C01810=1025.113,288.179,370.569,170.460,47.776,159.220
C01811=1025.106,287.931,370.600,170.455,47.778,159.220
C01812=1025.099,287.683,370.631,170.450,47.780,159.220
C01813=1025.092,287.435,370.663,170.446,47.782,159.220
C01814=1025.086,287.188,370.694,170.441,47.784,159.219
C01815=1025.080,286.940,370.725,170.437,47.786,159.219
C01816=1025.073,286.692,370.757,170.432,47.788,159.219
C01817=1025.066,286.444,370.788,170.428,47.790,159.219
C01818=1025.059,286.196,370.820,170.423,47.792,159.219
C01819=1025.053,285.948,370.851,170.419,47.794,159.219
C01820=1025.046,285.700,370.883,170.414,47.796,159.219
C01821=1025.039,285.452,370.914,170.410,47.798,159.218
C01822=1025.033,285.204,370.945,170.405,47.800,159.218
C01823=1025.026,284.956,370.976,170.400,47.802,159.218
C01824=1025.019,284.708,371.008,170.397,47.804,159.218
C01825=1025.013,284.461,371.039,170.392,47.806,159.218
C01826=1025.006,284.213,371.069,170.387,47.808,159.218
C01827=1024.999,283.965,371.100,170.382,47.810,159.217
C01828=1024.993,283.717,371.132,170.378,47.812,159.217
C01829=1024.986,283.468,371.162,170.374,47.814,159.217
C01830=1024.979,283.220,371.194,170.369,47.816,159.217
C01831=1024.973,282.973,371.225,170.365,47.818,159.217
C01832=1024.966,282.724,371.256,170.360,47.821,159.217
C01833=1024.959,282.477,371.286,170.356,47.823,159.217
C01834=1024.953,282.229,371.318,170.352,47.825,159.217
C01835=1024.946,281.981,371.349,170.347,47.827,159.216
C01836=1024.940,281.733,371.380,170.342,47.829,159.216
C01837=1024.933,281.484,371.411,170.339,47.831,159.216
C01838=1024.927,281.237,371.442,170.334,47.833,159.216
C01839=1024.920,280.989,371.473,170.329,47.835,159.216
C01840=1024.913,280.741,371.503,170.325,47.838,159.216
C01841=1024.906,280.493,371.535,170.321,47.839,159.216
C01842=1024.901,280.245,371.565,170.316,47.841,159.215
C01843=1024.894,279.997,371.597,170.312,47.844,159.216
C01844=1024.887,279.749,371.627,170.307,47.846,159.215
C01845=1024.880,279.501,371.658,170.303,47.848,159.215
C01846=1024.874,279.253,371.688,170.299,47.850,159.215
C01847=1024.867,279.005,371.720,170.294,47.853,159.215
C01848=1024.861,278.757,371.751,170.290,47.855,159.215
C01849=1024.851,278.345,371.802,170.283,47.858,159.215
C01850=1024.839,277.933,371.853,170.276,47.862,159.215
C01851=1024.829,277.521,371.904,170.269,47.866,159.215
C01852=1024.818,277.109,371.955,170.261,47.870,159.214
C01853=1024.811,276.860,371.985,170.256,47.872,159.214
C01854=1024.805,276.613,372.016,170.253,47.874,159.214
C01855=1024.798,276.365,372.047,170.248,47.876,159.214
C01856=1024.791,276.116,372.077,170.244,47.879,159.214
C01857=1024.785,275.869,372.107,170.239,47.881,159.214
C01858=1024.779,275.620,372.138,170.236,47.884,159.214
C01859=1024.771,275.372,372.169,170.231,47.886,159.214
C01860=1024.765,275.125,372.199,170.227,47.888,159.214
C01861=1024.758,274.876,372.229,170.222,47.891,159.214
C01862=1024.753,274.629,372.260,170.219,47.893,159.214
C01863=1024.746,274.380,372.290,170.214,47.895,159.214
C01864=1024.739,274.132,372.320,170.209,47.898,159.214
C01865=1024.733,273.884,372.351,170.206,47.900,159.213
C01866=1024.726,273.636,372.381,170.201,47.902,159.213
C01867=1024.720,273.388,372.411,170.197,47.905,159.213
C01868=1024.713,273.140,372.442,170.192,47.907,159.213
C01869=1024.706,272.892,372.473,170.189,47.910,159.213
C01870=1024.700,272.644,372.502,170.184,47.912,159.213
C01871=1024.693,272.396,372.533,170.180,47.914,159.213
C01872=1024.687,272.148,372.563,170.176,47.917,159.213
C01873=1024.681,271.899,372.593,170.172,47.919,159.213
C01874=1024.674,271.652,372.623,170.167,47.922,159.213
C01875=1024.668,271.403,372.653,170.163,47.924,159.213
C01876=1024.661,271.156,372.683,170.159,47.926,159.213
C01877=1024.655,270.907,372.714,170.155,47.929,159.213
C01878=1024.648,270.659,372.744,170.150,47.932,159.213
C01879=1024.642,270.411,372.774,170.147,47.934,159.213
C01880=1024.635,270.163,372.805,170.142,47.936,159.213
C01881=1024.629,269.915,372.835,170.138,47.939,159.213
C01882=1024.622,269.667,372.864,170.134,47.941,159.213
C01883=1024.615,269.419,372.894,170.130,47.944,159.213
C01884=1024.610,269.171,372.924,170.125,47.946,159.213
C01885=1024.602,268.923,372.954,170.121,47.949,159.213
C01886=1024.596,268.675,372.984,170.118,47.952,159.213
C01887=1024.590,268.426,373.014,170.113,47.954,159.213
C01888=1024.583,268.179,373.044,170.109,47.957,159.213
C01889=1024.576,267.930,373.074,170.105,47.959,159.213
C01890=1024.570,267.682,373.104,170.101,47.962,159.213
C01891=1024.563,267.434,373.134,170.096,47.964,159.213
C01892=1024.557,267.186,373.164,170.093,47.967,159.213
C01893=1024.550,266.937,373.193,170.088,47.969,159.213
C01894=1024.544,266.689,373.223,170.084,47.972,159.213
C01895=1024.538,266.442,373.253,170.080,47.975,159.213
C01896=1024.531,266.193,373.283,170.076,47.977,159.213
C01897=1024.525,265.945,373.313,170.072,47.980,159.213
C01898=1024.518,265.696,373.342,170.067,47.983,159.213
C01899=1024.511,265.449,373.372,170.064,47.985,159.213
C01900=1024.505,265.201,373.401,170.060,47.988,159.213
C01901=1024.498,264.953,373.431,170.055,47.991,159.213
C01902=1024.492,264.704,373.460,170.052,47.993,159.213
C01903=1024.485,264.456,373.491,170.047,47.996,159.213
C01904=1024.479,264.208,373.520,170.043,47.999,159.213
C01905=1024.468,263.801,373.569,170.036,48.003,159.213
C01906=1024.458,263.393,373.617,170.030,48.008,159.213
C01907=1024.448,262.986,373.665,170.023,48.012,159.213
C01908=1024.436,262.578,373.714,170.016,48.016,159.213
C01909=1024.430,262.330,373.744,170.013,48.019,159.213
C01910=1024.424,262.082,373.773,170.009,48.022,159.213
C01911=1024.417,261.834,373.803,170.004,48.025,159.213
C01912=1024.411,261.586,373.832,170.001,48.027,159.214
C01913=1024.404,261.337,373.861,169.996,48.030,159.214
C01914=1024.398,261.090,373.891,169.992,48.033,159.214
C01915=1024.391,260.841,373.920,169.989,48.035,159.214
C01916=1024.385,260.593,373.950,169.984,48.038,159.214
C01917=1024.378,260.345,373.979,169.980,48.041,159.214
C01918=1024.372,260.096,374.008,169.977,48.044,159.214
C01919=1024.365,259.848,374.038,169.972,48.047,159.214
C01920=1024.358,259.601,374.066,169.968,48.050,159.214
C01921=1024.352,259.352,374.095,169.964,48.053,159.214
C01922=1024.345,259.104,374.125,169.960,48.055,159.214
C01923=1024.339,258.856,374.154,169.956,48.059,159.214
C01924=1024.332,258.608,374.182,169.952,48.061,159.214
C01925=1024.325,258.360,374.211,169.948,48.065,159.214
C01926=1024.319,258.111,374.241,169.945,48.067,159.215
C01927=1024.312,257.863,374.270,169.940,48.070,159.215
C01928=1024.305,257.615,374.298,169.936,48.073,159.215
C01929=1024.298,257.366,374.327,169.933,48.076,159.215
C01930=1024.292,257.118,374.356,169.929,48.079,159.215
C01931=1024.286,256.870,374.385,169.924,48.082,159.215
C01932=1024.279,256.622,374.414,169.920,48.085,159.215
C01933=1024.273,256.374,374.443,169.917,48.088,159.215
C01934=1024.266,256.125,374.472,169.913,48.091,159.215
C01935=1024.259,255.876,374.500,169.908,48.094,159.215
C01936=1024.253,255.628,374.529,169.905,48.097,159.215
C01937=1024.247,255.380,374.558,169.901,48.100,159.216
C01938=1024.240,255.132,374.587,169.896,48.103,159.216
C01939=1024.233,254.884,374.616,169.892,48.106,159.216
C01940=1024.227,254.635,374.645,169.889,48.109,159.216
C01941=1024.220,254.387,374.674,169.885,48.112,159.216
C01942=1024.214,254.139,374.703,169.881,48.115,159.216
C01943=1024.207,253.891,374.731,169.877,48.118,159.216
C01944=1024.201,253.643,374.760,169.873,48.121,159.217
C01945=1024.194,253.394,374.789,169.869,48.124,159.217
C01946=1024.187,253.146,374.818,169.866,48.127,159.217
C01947=1024.181,252.898,374.847,169.862,48.130,159.217
C01948=1024.175,252.649,374.875,169.857,48.133,159.217
C01949=1024.169,252.401,374.904,169.854,48.136,159.217
C01950=1024.162,252.153,374.933,169.850,48.139,159.217
C01951=1024.156,251.904,374.961,169.846,48.143,159.217
C01952=1024.150,251.656,374.990,169.842,48.145,159.217
C01953=1024.143,251.408,375.018,169.839,48.149,159.218
C01954=1024.136,251.160,375.047,169.834,48.151,159.218
C01955=1024.131,250.912,375.076,169.830,48.155,159.218
C01956=1024.124,250.663,375.105,169.827,48.158,159.218
C01957=1024.117,250.415,375.134,169.823,48.161,159.218
C01958=1024.111,250.166,375.162,169.819,48.164,159.218
C01959=1024.105,249.918,375.191,169.815,48.167,159.218
C01960=1024.098,249.670,375.219,169.811,48.170,159.218
C01961=1024.088,249.261,375.266,169.805,48.176,159.219
C01962=1024.077,248.852,375.313,169.799,48.180,159.219
C01963=1024.067,248.442,375.361,169.792,48.186,159.219
C01964=1024.057,248.034,375.407,169.786,48.191,159.219
C01965=1024.050,247.786,375.436,169.783,48.194,159.220
C01966=1024.044,247.538,375.465,169.778,48.197,159.220
C01967=1024.037,247.289,375.493,169.775,48.200,159.220
C01968=1024.031,247.041,375.522,169.771,48.203,159.220
C01969=1024.025,246.792,375.550,169.767,48.207,159.220
C01970=1024.018,246.544,375.579,169.764,48.209,159.220
C01971=1024.012,246.296,375.607,169.760,48.213,159.221
C01972=1024.006,246.047,375.636,169.756,48.216,159.221
C01973=1023.999,245.799,375.664,169.753,48.219,159.221
C01974=1023.993,245.551,375.693,169.748,48.222,159.221
C01975=1023.987,245.302,375.721,169.744,48.225,159.221
C01976=1023.981,245.053,375.749,169.741,48.228,159.221
C01977=1023.975,244.806,375.778,169.737,48.232,159.222
C01978=1023.969,244.558,375.806,169.734,48.235,159.222
C01979=1023.963,244.309,375.835,169.729,48.238,159.222
C01980=1023.956,244.061,375.863,169.725,48.241,159.222
C01981=1023.950,243.812,375.891,169.722,48.244,159.222
C01982=1023.943,243.564,375.919,169.718,48.248,159.222
C01983=1023.937,243.316,375.948,169.714,48.251,159.223
C01984=1023.930,243.067,375.975,169.711,48.254,159.223
C01985=1023.925,242.820,376.004,169.707,48.258,159.223
C01986=1023.918,242.571,376.032,169.703,48.261,159.223
C01987=1023.912,242.323,376.060,169.700,48.264,159.223
C01988=1023.905,242.074,376.088,169.696,48.268,159.224
C01989=1023.899,241.826,376.116,169.692,48.271,159.224
C01990=1023.893,241.578,376.145,169.689,48.274,159.224
C01991=1023.886,241.329,376.172,169.685,48.278,159.224
C01992=1023.880,241.080,376.201,169.681,48.281,159.224
C01993=1023.874,240.833,376.228,169.678,48.284,159.225
C01994=1023.867,240.584,376.256,169.674,48.288,159.225
C01995=1023.861,240.335,376.284,169.670,48.291,159.225
C01996=1023.855,240.087,376.312,169.667,48.294,159.225
C01997=1023.848,239.839,376.341,169.662,48.298,159.225
C01998=1023.842,239.591,376.368,169.658,48.301,159.226
C01999=1023.836,239.343,376.396,169.655,48.304,159.226
C02000=1023.829,239.094,376.424,169.652,48.309,159.226
C02001=1023.822,238.846,376.452,169.648,48.312,159.226
C02002=1023.816,238.597,376.480,169.645,48.315,159.227
C02003=1023.810,238.349,376.508,169.640,48.319,159.227
C02004=1023.804,238.100,376.534,169.637,48.323,159.227
C02005=1023.797,237.852,376.562,169.634,48.326,159.227
C02006=1023.790,237.603,376.590,169.630,48.329,159.228
C02007=1023.784,237.355,376.617,169.626,48.333,159.228
C02008=1023.778,237.107,376.645,169.623,48.336,159.228
C02009=1023.772,236.858,376.673,169.619,48.340,159.228
C02010=1023.765,236.610,376.701,169.615,48.343,159.228
C02011=1023.758,236.362,376.729,169.611,48.347,159.229
C02012=1023.752,236.113,376.756,169.608,48.351,159.229
C02013=1023.746,235.865,376.783,169.604,48.354,159.229
C02014=1023.739,235.616,376.811,169.600,48.358,159.229
C02015=1023.733,235.368,376.838,169.597,48.361,159.230
C02016=1023.726,235.119,376.866,169.593,48.365,159.230
C02017=1023.716,234.704,376.912,169.587,48.370,159.230
C02018=1023.705,234.289,376.958,169.581,48.377,159.231
C02019=1023.694,233.874,377.004,169.574,48.383,159.231
C02020=1023.684,233.458,377.050,169.569,48.388,159.232
C02021=1023.678,233.210,377.077,169.565,48.392,159.232
C02022=1023.671,232.962,377.105,169.561,48.396,159.232
C02023=1023.665,232.713,377.132,169.559,48.400,159.233
C02024=1023.658,232.464,377.160,169.555,48.403,159.233
C02025=1023.652,232.217,377.187,169.550,48.407,159.233
C02026=1023.646,231.968,377.214,169.548,48.410,159.233
C02027=1023.639,231.719,377.242,169.544,48.414,159.234
C02028=1023.633,231.471,377.269,169.540,48.418,159.234
C02029=1023.627,231.222,377.296,169.536,48.421,159.234
C02030=1023.620,230.975,377.324,169.533,48.425,159.234
C02031=1023.614,230.726,377.351,169.529,48.429,159.235
C02032=1023.607,230.477,377.378,169.525,48.432,159.235
C02033=1023.601,230.229,377.406,169.522,48.436,159.235
C02034=1023.595,229.980,377.433,169.518,48.439,159.235
C02035=1023.588,229.732,377.461,169.515,48.444,159.236
C02036=1023.582,229.484,377.487,169.512,48.447,159.236
C02037=1023.576,229.235,377.515,169.508,48.451,159.236
C02038=1023.570,228.987,377.542,169.504,48.455,159.237
C02039=1023.563,228.738,377.569,169.501,48.458,159.237
C02040=1023.557,228.489,377.596,169.497,48.462,159.237
C02041=1023.551,228.241,377.624,169.493,48.466,159.238
C02042=1023.545,227.992,377.651,169.491,48.470,159.238
C02043=1023.538,227.745,377.678,169.487,48.474,159.238
C02044=1023.531,227.496,377.705,169.483,48.477,159.239
C02045=1023.525,227.247,377.732,169.479,48.481,159.239
C02046=1023.519,226.999,377.759,169.476,48.485,159.239
C02047=1023.512,226.750,377.786,169.472,48.489,159.239
C02048=1023.506,226.502,377.812,169.469,48.493,159.240
C02049=1023.499,226.254,377.840,169.466,48.496,159.240
C02050=1023.494,226.005,377.866,169.462,48.500,159.240
C02051=1023.486,225.756,377.893,169.458,48.504,159.241
C02052=1023.480,225.508,377.921,169.455,48.508,159.241
C02053=1023.474,225.260,377.947,169.452,48.512,159.242
C02054=1023.467,225.011,377.974,169.448,48.516,159.242
C02055=1023.461,224.763,378.000,169.444,48.520,159.242
C02056=1023.454,224.514,378.028,169.440,48.524,159.242
C02057=1023.448,224.266,378.054,169.438,48.528,159.243
C02058=1023.441,224.017,378.081,169.434,48.532,159.243
C02059=1023.436,223.769,378.108,169.430,48.536,159.244
C02060=1023.429,223.520,378.134,169.426,48.539,159.244
C02061=1023.423,223.272,378.161,169.423,48.543,159.244
C02062=1023.416,223.023,378.188,169.420,48.547,159.244
C02063=1023.410,222.775,378.215,169.416,48.551,159.245
C02064=1023.403,222.526,378.242,169.413,48.555,159.245
C02065=1023.397,222.278,378.268,169.410,48.559,159.246
C02066=1023.390,222.029,378.295,169.406,48.563,159.246
C02067=1023.385,221.780,378.321,169.402,48.567,159.246
C02068=1023.378,221.532,378.349,169.399,48.571,159.247
C02069=1023.371,221.284,378.375,169.395,48.575,159.247
C02070=1023.365,221.035,378.402,169.392,48.579,159.247
C02071=1023.359,220.787,378.429,169.389,48.583,159.248
C02072=1023.352,220.538,378.455,169.385,48.587,159.248
C02073=1023.347,220.326,378.478,169.382,48.590,159.248
C02074=1023.342,220.115,378.500,169.379,48.593,159.249
C02075=1023.336,219.903,378.523,169.377,48.597,159.249
C02076=1023.332,219.691,378.546,169.374,48.600,159.249
C02077=1023.326,219.481,378.569,169.371,48.604,159.249
C02078=1023.320,219.269,378.591,169.368,48.607,159.250
C02079=1023.316,219.057,378.614,169.365,48.611,159.250
C02080=1023.310,218.846,378.636,169.362,48.614,159.250
C02081=1023.304,218.597,378.663,169.358,48.618,159.251
C02082=1023.297,218.349,378.690,169.355,48.623,159.251
C02083=1023.290,218.100,378.716,169.351,48.627,159.252
C02084=1023.284,217.852,378.743,169.348,48.631,159.252
C02085=1023.278,217.603,378.768,169.345,48.635,159.252
C02086=1023.271,217.354,378.794,169.341,48.639,159.253
C02087=1023.265,217.106,378.821,169.337,48.643,159.253
C02088=1023.258,216.857,378.847,169.335,48.647,159.253
C02089=1023.252,216.609,378.873,169.331,48.651,159.254
C02090=1023.246,216.361,378.900,169.327,48.655,159.254
C02091=1023.239,216.111,378.926,169.324,48.660,159.255
C02092=1023.232,215.863,378.952,169.321,48.664,159.255
C02093=1023.226,215.614,378.979,169.317,48.668,159.255
C02094=1023.220,215.366,379.005,169.314,48.672,159.256
C02095=1023.214,215.118,379.032,169.310,48.676,159.256
C02096=1023.207,214.868,379.057,169.307,48.680,159.257
C02097=1023.200,214.620,379.083,169.304,48.685,159.257
C02098=1023.195,214.372,379.110,169.300,48.689,159.257
C02099=1023.188,214.123,379.136,169.297,48.693,159.258
C02100=1023.181,213.875,379.162,169.293,48.697,159.258
C02101=1023.176,213.626,379.188,169.290,48.701,159.259
C02102=1023.169,213.377,379.215,169.287,48.706,159.259
C02103=1023.162,213.129,379.240,169.283,48.710,159.259
C02104=1023.157,212.880,379.267,169.279,48.714,159.260
C02105=1023.150,212.632,379.293,169.277,48.718,159.260
C02106=1023.143,212.384,379.319,169.273,48.723,159.261
C02107=1023.137,212.135,379.345,169.270,48.727,159.261
C02108=1023.131,211.887,379.371,169.266,48.731,159.261
C02109=1023.125,211.637,379.398,169.263,48.735,159.262
C02110=1023.118,211.389,379.424,169.260,48.740,159.262
C02111=1023.112,211.141,379.450,169.256,48.744,159.263
C02112=1023.106,210.892,379.476,169.252,48.748,159.263
C02113=1023.099,210.643,379.502,169.250,48.752,159.264
C02114=1023.093,210.395,379.528,169.246,48.757,159.264
C02115=1023.087,210.146,379.554,169.243,48.761,159.264
C02116=1023.081,209.898,379.580,169.239,48.765,159.265
C02117=1023.074,209.649,379.606,169.237,48.770,159.265
C02118=1023.067,209.401,379.632,169.233,48.774,159.266
C02119=1023.061,209.152,379.657,169.230,48.779,159.266
C02120=1023.055,208.904,379.683,169.226,48.783,159.267
C02121=1023.048,208.655,379.709,169.223,48.788,159.267
C02122=1023.042,208.406,379.736,169.220,48.792,159.268
C02123=1023.036,208.157,379.761,169.216,48.796,159.268
C02124=1023.029,207.909,379.787,169.213,48.801,159.268
C02125=1023.023,207.661,379.812,169.209,48.805,159.269
C02126=1023.016,207.411,379.838,169.207,48.809,159.269
C02127=1023.010,207.163,379.864,169.203,48.814,159.270
C02128=1023.004,206.915,379.889,169.200,48.818,159.270
C02129=1022.997,206.667,379.915,169.196,48.823,159.271
C02130=1022.991,206.418,379.941,169.193,48.827,159.271
C02131=1022.985,206.168,379.967,169.190,48.831,159.272
C02132=1022.978,205.920,379.993,169.187,48.836,159.272
C02133=1022.968,205.500,380.036,169.181,48.844,159.273
C02134=1022.957,205.080,380.080,169.175,48.851,159.274
C02135=1022.946,204.659,380.122,169.169,48.859,159.274
C02136=1022.935,204.239,380.166,169.164,48.867,159.275
C02137=1022.911,203.207,380.265,168.742,48.769,159.192
C02138=1022.906,202.959,380.290,168.738,48.774,159.192
C02139=1022.900,202.709,380.314,168.734,48.780,159.193
C02140=1022.895,202.460,380.338,168.730,48.785,159.193
C02141=1022.889,202.212,380.361,168.725,48.790,159.194
C02142=1022.884,201.963,380.386,168.721,48.796,159.194
C02143=1022.879,201.715,380.410,168.717,48.801,159.195
C02144=1022.873,201.465,380.434,168.713,48.807,159.196
C02145=1022.867,201.216,380.458,168.708,48.812,159.196
C02146=1022.862,200.968,380.482,168.705,48.818,159.197
C02147=1022.856,200.719,380.506,168.701,48.823,159.197
C02148=1022.851,200.470,380.530,168.696,48.828,159.197
C02149=1022.845,200.222,380.553,168.692,48.834,159.198
C02150=1022.839,199.973,380.578,168.688,48.839,159.198
C02151=1022.834,199.723,380.601,168.684,48.845,159.199
C02152=1022.828,199.475,380.625,168.680,48.850,159.199
C02153=1022.823,199.226,380.649,168.675,48.856,159.200
C02154=1022.817,198.978,380.672,168.671,48.861,159.200
C02155=1022.812,198.729,380.695,168.667,48.867,159.201
C02156=1022.806,198.479,380.720,168.663,48.873,159.202
C02157=1022.800,198.230,380.743,168.659,48.878,159.202
C02158=1022.795,197.982,380.767,168.655,48.884,159.203
C02159=1022.789,197.733,380.790,168.651,48.890,159.203
C02160=1022.783,197.485,380.814,168.646,48.895,159.204
C02161=1022.778,197.236,380.837,168.642,48.901,159.204
C02162=1022.772,196.987,380.861,168.638,48.906,159.205
C02163=1022.766,196.738,380.884,168.634,48.912,159.205
C02164=1022.761,196.489,380.907,168.630,48.917,159.206
C02165=1022.754,196.240,380.931,168.625,48.923,159.206
C02166=1022.749,195.991,380.955,168.621,48.928,159.207
C02167=1022.743,195.743,380.979,168.617,48.934,159.207
C02168=1022.738,195.494,381.002,168.613,48.939,159.208
C02169=1022.733,195.245,381.025,168.609,48.945,159.208
C02170=1022.727,194.996,381.049,168.606,48.951,159.209
C02171=1022.721,194.747,381.072,168.601,48.956,159.210
C02172=1022.716,194.498,381.095,168.597,48.962,159.210
C02173=1022.710,194.250,381.119,168.593,48.968,159.211
C02174=1022.705,194.001,381.142,168.589,48.973,159.211
C02175=1022.699,193.752,381.165,168.585,48.979,159.212
C02176=1022.693,193.504,381.189,168.581,48.985,159.212
C02177=1022.688,193.254,381.213,168.576,48.990,159.213
C02178=1022.682,193.005,381.236,168.572,48.996,159.213
C02179=1022.677,192.757,381.258,168.568,49.001,159.214
C02180=1022.671,192.508,381.283,168.565,49.006,159.214
C02181=1022.666,192.259,381.306,168.561,49.012,159.215
C02182=1022.660,192.010,381.329,168.557,49.018,159.216
C02183=1022.655,191.761,381.352,168.553,49.023,159.216
C02184=1022.649,191.512,381.375,168.548,49.029,159.217
C02185=1022.644,191.263,381.399,168.544,49.035,159.217
C02186=1022.638,191.015,381.422,168.541,49.040,159.218
C02187=1022.632,190.766,381.445,168.537,49.046,159.218
C02188=1022.627,190.516,381.469,168.533,49.052,159.219
C02189=1022.622,190.268,381.492,168.529,49.057,159.219
C02190=1022.616,190.019,381.515,168.525,49.063,159.220
C02191=1022.611,189.771,381.539,168.521,49.068,159.221
C02192=1022.606,189.522,381.562,168.517,49.073,159.221
C02193=1022.600,189.273,381.584,168.513,49.079,159.222
C02194=1022.595,189.024,381.608,168.509,49.085,159.222
C02195=1022.589,188.775,381.631,168.505,49.090,159.223
C02196=1022.583,188.526,381.654,168.501,49.096,159.223
C02197=1022.578,188.277,381.677,168.498,49.102,159.224
C02198=1022.572,187.995,381.704,168.493,49.108,159.224
C02199=1022.566,187.713,381.730,168.488,49.115,159.225
C02200=1022.560,187.431,381.756,168.484,49.121,159.226
C02201=1022.554,187.150,381.782,168.479,49.128,159.226
C02202=1022.548,186.901,381.805,168.476,49.132,159.227
C02203=1022.543,186.652,381.828,168.472,49.138,159.227
C02204=1022.538,186.403,381.851,168.468,49.144,159.228
C02205=1022.532,186.154,381.874,168.464,49.149,159.228
C02206=1022.527,185.905,381.898,168.461,49.155,159.229
C02207=1022.522,185.656,381.920,168.457,49.161,159.230
C02208=1022.516,185.408,381.943,168.453,49.167,159.230
C02209=1022.511,185.158,381.967,168.448,49.172,159.231
C02210=1022.505,184.909,381.990,168.445,49.177,159.231
C02211=1022.500,184.661,382.012,168.441,49.183,159.232
C02212=1022.495,184.412,382.036,168.437,49.189,159.232
C02213=1022.489,184.163,382.059,168.434,49.194,159.233
C02214=1022.484,183.914,382.082,168.430,49.200,159.234
C02215=1022.479,183.664,382.105,168.426,49.206,159.234
C02216=1022.474,183.416,382.127,168.421,49.211,159.235
C02217=1022.468,183.167,382.150,168.419,49.217,159.235
C02218=1022.463,182.918,382.174,168.414,49.223,159.236
C02219=1022.457,182.669,382.197,168.410,49.228,159.236
C02220=1022.452,182.421,382.219,168.407,49.233,159.237
C02221=1022.447,182.172,382.241,168.403,49.239,159.238
C02222=1022.441,181.923,382.264,168.399,49.245,159.238
C02223=1022.436,181.673,382.287,168.395,49.251,159.239
C02224=1022.430,181.424,382.310,168.391,49.257,159.239
C02225=1022.424,181.176,382.331,168.388,49.263,159.240
C02226=1022.419,180.927,382.354,168.384,49.269,159.241
C02227=1022.413,180.678,382.377,168.380,49.274,159.241
C02228=1022.407,180.429,382.398,168.376,49.280,159.242
C02229=1022.402,180.181,382.421,168.372,49.286,159.242
C02230=1022.396,179.931,382.443,168.369,49.292,159.243
C02231=1022.391,179.682,382.466,168.366,49.298,159.244
C02232=1022.384,179.433,382.488,168.362,49.304,159.244
C02233=1022.380,179.184,382.510,168.358,49.310,159.245
C02234=1022.374,178.935,382.533,168.354,49.316,159.246
C02235=1022.368,178.686,382.554,168.351,49.322,159.246
C02236=1022.362,178.437,382.577,168.347,49.328,159.247
C02237=1022.357,178.188,382.599,168.343,49.334,159.247
C02238=1022.351,177.940,382.621,168.339,49.339,159.248
C02239=1022.345,177.690,382.644,168.336,49.345,159.249
C02240=1022.340,177.442,382.666,168.332,49.351,159.249
C02241=1022.334,177.193,382.688,168.328,49.357,159.250
C02242=1022.329,176.943,382.710,168.324,49.363,159.250
C02243=1022.323,176.695,382.733,168.321,49.368,159.251
C02244=1022.318,176.446,382.755,168.317,49.374,159.252
C02245=1022.312,176.196,382.776,168.313,49.380,159.252
C02246=1022.307,175.948,382.799,168.309,49.386,159.253
C02247=1022.301,175.699,382.821,168.306,49.392,159.253
C02248=1022.295,175.449,382.843,168.302,49.398,159.254
C02249=1022.290,175.201,382.866,168.298,49.404,159.255
C02250=1022.285,174.952,382.888,168.295,49.410,159.256
C02251=1022.279,174.703,382.909,168.291,49.416,159.256
C02252=1022.273,174.454,382.932,168.287,49.422,159.257
C02253=1022.268,174.205,382.954,168.283,49.428,159.257
C02254=1022.262,173.956,382.975,168.280,49.433,159.258
C02255=1022.257,173.707,382.998,168.276,49.439,159.259
C02256=1022.252,173.459,383.020,168.272,49.445,159.259
C02257=1022.246,173.209,383.042,168.269,49.451,159.260
C02258=1022.240,172.960,383.064,168.265,49.457,159.260
C02259=1022.235,172.712,383.087,168.261,49.463,159.261
C02260=1022.229,172.462,383.108,168.258,49.468,159.262
C02261=1022.224,172.214,383.130,168.254,49.474,159.262
C02262=1022.215,171.810,383.166,168.249,49.484,159.263
C02263=1022.207,171.405,383.202,168.243,49.493,159.264
C02264=1022.199,171.076,383.231,168.238,49.501,159.265
C02265=1022.192,170.746,383.260,168.234,49.509,159.266
C02266=1022.185,170.418,383.289,168.228,49.517,159.267
C02267=1022.178,170.088,383.319,168.224,49.525,159.268
C02268=1022.172,169.839,383.340,168.220,49.530,159.268
C02269=1022.167,169.590,383.362,168.217,49.536,159.269
C02270=1022.162,169.341,383.384,168.213,49.542,159.269
C02271=1022.156,169.092,383.406,168.209,49.548,159.270
C02272=1022.151,168.843,383.428,168.206,49.554,159.271
C02273=1022.145,168.594,383.450,168.202,49.560,159.271
C02274=1022.140,168.345,383.472,168.199,49.565,159.272
C02275=1022.134,168.096,383.494,168.195,49.571,159.273
C02276=1022.129,167.847,383.515,168.191,49.577,159.273
C02277=1022.124,167.599,383.537,168.189,49.583,159.274
C02278=1022.118,167.349,383.559,168.185,49.589,159.275
C02279=1022.113,167.101,383.580,168.182,49.595,159.275
C02280=1022.107,166.851,383.603,168.178,49.601,159.276
C02281=1022.103,166.602,383.625,168.175,49.607,159.276
C02282=1022.096,166.353,383.646,168.171,49.613,159.277
C02283=1022.092,166.104,383.668,168.167,49.619,159.278
C02284=1022.087,165.855,383.690,168.164,49.624,159.278
C02285=1022.081,165.606,383.712,168.160,49.630,159.279
C02286=1022.076,165.357,383.733,168.157,49.636,159.280
C02287=1022.070,165.108,383.756,168.153,49.642,159.280
C02288=1022.065,164.859,383.777,168.150,49.647,159.281
C02289=1022.060,164.611,383.799,168.146,49.653,159.281
C02290=1022.054,164.361,383.821,168.143,49.659,159.282
C02291=1022.049,164.113,383.842,168.139,49.665,159.283
C02292=1022.044,163.864,383.864,168.136,49.671,159.283
C02293=1022.039,163.614,383.886,168.132,49.677,159.284
C02294=1022.033,163.366,383.908,168.129,49.682,159.285
C02295=1022.028,163.117,383.930,168.126,49.688,159.285
C02296=1022.022,162.868,383.951,168.123,49.695,159.286
C02297=1022.018,162.618,383.972,168.119,49.701,159.287
C02298=1022.013,162.369,383.994,168.116,49.706,159.287
C02299=1022.007,162.120,384.016,168.112,49.712,159.288
C02300=1022.002,161.871,384.038,168.109,49.718,159.288
C02301=1021.997,161.623,384.060,168.105,49.724,159.289
C02302=1021.991,161.373,384.081,168.102,49.730,159.290
C02303=1021.986,161.125,384.103,168.098,49.736,159.290
C02304=1021.981,160.875,384.124,168.095,49.741,159.291
C02305=1021.975,160.626,384.146,168.091,49.747,159.292
C02306=1021.970,160.377,384.168,168.089,49.753,159.292
C02307=1021.965,160.129,384.189,168.085,49.759,159.293
C02308=1021.960,159.880,384.211,168.082,49.764,159.293
C02309=1021.955,159.630,384.232,168.078,49.770,159.294
C02310=1021.949,159.381,384.254,168.075,49.776,159.295
C02311=1021.945,159.132,384.275,168.072,49.782,159.295
C02312=1021.939,158.884,384.297,168.068,49.788,159.296
C02313=1021.934,158.634,384.318,168.065,49.793,159.297
C02314=1021.928,158.385,384.340,168.061,49.800,159.297
C02315=1021.923,158.136,384.360,168.057,49.806,159.298
C02316=1021.917,157.887,384.382,168.055,49.812,159.299
C02317=1021.911,157.638,384.403,168.051,49.818,159.299
C02318=1021.907,157.389,384.424,168.048,49.824,159.300
C02319=1021.901,157.140,384.446,168.044,49.830,159.301
C02320=1021.895,156.891,384.466,168.041,49.836,159.301
C02321=1021.890,156.642,384.488,168.038,49.843,159.302
C02322=1021.885,156.393,384.508,168.035,49.848,159.303
C02323=1021.878,156.144,384.530,168.031,49.854,159.303
C02324=1021.873,155.861,384.553,168.027,49.861,159.304
C02325=1021.867,155.578,384.577,168.024,49.868,159.305
C02326=1021.860,155.296,384.602,168.019,49.875,159.305
C02327=1021.855,155.013,384.625,168.016,49.881,159.306
C02328=1021.849,154.765,384.646,168.013,49.888,159.307
C02329=1021.844,154.514,384.668,168.009,49.894,159.308
C02330=1021.839,154.265,384.688,168.006,49.899,159.308
C02331=1021.833,154.017,384.710,168.002,49.905,159.309
C02332=1021.828,153.768,384.730,168.000,49.912,159.310
C02333=1021.822,153.518,384.752,167.996,49.918,159.310
C02334=1021.816,153.269,384.772,167.993,49.923,159.311
C02335=1021.812,153.020,384.794,167.989,49.930,159.312
C02336=1021.806,152.771,384.815,167.986,49.936,159.312
C02337=1021.801,152.522,384.835,167.982,49.942,159.313
C02338=1021.795,152.272,384.856,167.980,49.947,159.314
C02339=1021.790,152.024,384.878,167.976,49.954,159.314
C02340=1021.784,151.775,384.898,167.973,49.960,159.315
C02341=1021.779,151.526,384.919,167.969,49.966,159.316
C02342=1021.774,151.277,384.940,167.967,49.972,159.317
C02343=1021.768,151.028,384.960,167.963,49.978,159.317
C02344=1021.762,150.778,384.981,167.960,49.984,159.318
C02345=1021.757,150.529,385.002,167.956,49.991,159.319
C02346=1021.752,150.281,385.023,167.953,49.996,159.319
C02347=1021.746,150.031,385.044,167.949,50.002,159.320
C02348=1021.741,149.782,385.064,167.947,50.009,159.321
C02349=1021.736,149.533,385.085,167.944,50.015,159.321
C02350=1021.730,149.285,385.106,167.940,50.021,159.322
C02351=1021.724,149.035,385.127,167.937,50.026,159.323
C02352=1021.719,148.786,385.148,167.934,50.033,159.323
C02353=1021.714,148.537,385.168,167.931,50.039,159.324
C02354=1021.709,148.288,385.189,167.927,50.045,159.325
C02355=1021.703,148.039,385.210,167.924,50.051,159.325
C02356=1021.698,147.790,385.231,167.920,50.057,159.326
C02357=1021.693,147.541,385.251,167.918,50.063,159.327
C02358=1021.687,147.292,385.272,167.914,50.070,159.327
C02359=1021.681,147.043,385.292,167.911,50.075,159.328
C02360=1021.676,146.794,385.312,167.908,50.081,159.329
C02361=1021.670,146.544,385.333,167.905,50.088,159.330
C02362=1021.665,146.295,385.354,167.902,50.093,159.330
C02363=1021.660,146.046,385.374,167.898,50.099,159.331
C02364=1021.654,145.797,385.395,167.895,50.106,159.332
C02365=1021.649,145.548,385.416,167.891,50.112,159.332
C02366=1021.644,145.299,385.437,167.889,50.118,159.333
C02367=1021.638,145.050,385.457,167.885,50.124,159.334
C02368=1021.633,144.800,385.476,167.882,50.130,159.334
C02369=1021.627,144.551,385.497,167.880,50.136,159.335
C02370=1021.621,144.302,385.517,167.876,50.143,159.336
C02371=1021.616,144.053,385.537,167.873,50.149,159.337
C02372=1021.611,143.804,385.558,167.869,50.155,159.337
C02373=1021.606,143.555,385.579,167.866,50.161,159.338
C02374=1021.600,143.306,385.598,167.863,50.167,159.339
C02375=1021.594,143.057,385.619,167.860,50.173,159.339
C02376=1021.589,142.808,385.640,167.857,50.180,159.340
C02377=1021.584,142.559,385.660,167.854,50.186,159.341
C02378=1021.577,142.309,385.680,167.851,50.191,159.341
C02379=1021.572,142.060,385.701,167.847,50.198,159.342
C02380=1021.567,141.811,385.722,167.844,50.204,159.343
C02381=1021.562,141.562,385.742,167.841,50.211,159.344
C02382=1021.556,141.313,385.761,167.838,50.216,159.344
C02383=1021.551,141.063,385.782,167.835,50.222,159.345
C02384=1021.545,140.814,385.802,167.832,50.229,159.346
C02385=1021.540,140.566,385.822,167.829,50.235,159.346
C02386=1021.535,140.317,385.843,167.825,50.241,159.347
C02387=1021.529,140.068,385.863,167.822,50.247,159.348
C02388=1021.523,139.784,385.886,167.819,50.254,159.348
C02389=1021.517,139.502,385.909,167.815,50.261,159.349
C02390=1021.511,139.219,385.932,167.812,50.267,159.350
C02391=1021.505,138.936,385.955,167.809,50.275,159.351
C02392=1021.500,138.687,385.976,167.805,50.281,159.352
C02393=1021.494,138.437,385.995,167.802,50.287,159.352
C02394=1021.489,138.188,386.015,167.798,50.293,159.353
C02395=1021.484,137.939,386.036,167.796,50.299,159.354
C02396=1021.478,137.690,386.055,167.793,50.305,159.354
C02397=1021.473,137.441,386.076,167.789,50.312,159.355
C02398=1021.467,137.192,386.096,167.787,50.318,159.356
C02399=1021.461,136.943,386.116,167.783,50.324,159.356
C02400=1021.456,136.693,386.136,167.780,50.330,159.357
C02401=1021.450,136.444,386.156,167.778,50.336,159.358
C02402=1021.445,136.195,386.177,167.774,50.342,159.359
C02403=1021.439,135.946,386.196,167.771,50.349,159.359
C02404=1021.434,135.696,386.216,167.767,50.355,159.360
C02405=1021.429,135.447,386.236,167.765,50.361,159.361
C02406=1021.424,135.199,386.256,167.762,50.367,159.361
C02407=1021.418,134.950,386.276,167.758,50.374,159.362
C02408=1021.412,134.700,386.295,167.756,50.380,159.363
C02409=1021.407,134.451,386.316,167.753,50.385,159.364
C02410=1021.401,134.202,386.335,167.749,50.392,159.364
C02411=1021.396,133.953,386.355,167.746,50.398,159.365
C02412=1021.390,133.703,386.375,167.743,50.405,159.366
C02413=1021.385,133.454,386.395,167.740,50.410,159.366
C02414=1021.379,133.205,386.415,167.738,50.417,159.367
C02415=1021.375,132.956,386.435,167.734,50.423,159.368
C02416=1021.369,132.707,386.455,167.731,50.429,159.369
C02417=1021.364,132.458,386.474,167.728,50.435,159.369
C02418=1021.358,132.209,386.494,167.725,50.442,159.370
C02419=1021.353,131.959,386.514,167.722,50.448,159.371
C02420=1021.347,131.710,386.534,167.719,50.453,159.371
C02421=1021.342,131.462,386.553,167.716,50.460,159.372
C02422=1021.337,131.212,386.574,167.713,50.466,159.373
C02423=1021.331,130.963,386.593,167.711,50.472,159.374
C02424=1021.326,130.714,386.613,167.707,50.479,159.374
C02425=1021.320,130.464,386.633,167.704,50.484,159.375
C02426=1021.315,130.215,386.653,167.701,50.491,159.376
C02427=1021.310,129.967,386.672,167.697,50.497,159.376
C02428=1021.304,129.717,386.691,167.695,50.503,159.377
C02429=1021.298,129.468,386.711,167.691,50.509,159.378
C02430=1021.293,129.219,386.731,167.689,50.516,159.379
C02431=1021.287,128.969,386.750,167.686,50.522,159.380
C02432=1021.282,128.720,386.770,167.682,50.528,159.380
C02433=1021.276,128.472,386.789,167.680,50.535,159.381
C02434=1021.270,128.222,386.808,167.676,50.541,159.382
C02435=1021.265,127.973,386.828,167.674,50.548,159.382
C02436=1021.259,127.723,386.847,167.671,50.554,159.383
C02437=1021.253,127.475,386.867,167.667,50.560,159.384
C02438=1021.248,127.226,386.886,167.665,50.567,159.385
C02439=1021.243,126.976,386.906,167.661,50.573,159.385
C02440=1021.237,126.727,386.925,167.659,50.579,159.386
C02441=1021.232,126.477,386.944,167.656,50.585,159.387
C02442=1021.226,126.228,386.964,167.652,50.592,159.388
C02443=1021.221,125.980,386.983,167.650,50.598,159.388
C02444=1021.215,125.730,387.002,167.647,50.604,159.389
C02445=1021.209,125.481,387.021,167.644,50.611,159.390
C02446=1021.204,125.231,387.041,167.641,50.617,159.390
C02447=1021.198,124.983,387.060,167.637,50.623,159.391
C02448=1021.193,124.734,387.080,167.635,50.629,159.392
C02449=1021.187,124.484,387.099,167.632,50.636,159.393
C02450=1021.182,124.235,387.119,167.628,50.642,159.393
C02451=1021.177,123.986,387.137,167.626,50.648,159.394
C02452=1021.170,123.702,387.160,167.622,50.655,159.395
C02453=1021.163,123.420,387.181,167.619,50.663,159.396
C02454=1021.158,123.137,387.203,167.616,50.669,159.397
C02455=1021.152,122.854,387.225,167.613,50.677,159.398
C02456=1021.146,122.604,387.244,167.609,50.683,159.398
C02457=1021.140,122.355,387.264,167.607,50.690,159.399
C02458=1021.135,122.106,387.282,167.604,50.695,159.400
C02459=1021.129,121.857,387.302,167.601,50.702,159.401
C02460=1021.123,121.608,387.322,167.597,50.708,159.401
C02461=1021.119,121.359,387.341,167.595,50.714,159.402
C02462=1021.113,121.109,387.360,167.592,50.720,159.403
C02463=1021.108,120.860,387.380,167.589,50.727,159.403
C02464=1021.103,120.611,387.399,167.586,50.733,159.404
C02465=1021.097,120.362,387.418,167.584,50.739,159.405
C02466=1021.091,120.112,387.437,167.580,50.746,159.405
C02467=1021.086,119.864,387.456,167.577,50.752,159.406
C02468=1021.080,119.614,387.475,167.574,50.758,159.407
C02469=1021.075,119.365,387.494,167.572,50.764,159.408
C02470=1021.070,119.116,387.513,167.568,50.771,159.408
C02471=1021.064,118.867,387.532,167.565,50.776,159.409
C02472=1021.059,118.617,387.552,167.563,50.783,159.410
C02473=1021.054,118.368,387.571,167.559,50.789,159.410
C02474=1021.048,118.119,387.590,167.557,50.795,159.411
C02475=1021.043,117.869,387.610,167.554,50.801,159.412
C02476=1021.038,117.621,387.629,167.552,50.808,159.413
C02477=1021.032,117.371,387.648,167.548,50.814,159.413
C02478=1021.027,117.122,387.667,167.545,50.820,159.414
C02479=1021.021,116.873,387.686,167.543,50.826,159.415
C02480=1021.015,116.624,387.705,167.540,50.833,159.416
C02481=1021.010,116.375,387.724,167.536,50.839,159.416
C02482=1021.005,116.125,387.743,167.534,50.845,159.417
C02483=1021.000,115.877,387.762,167.531,50.851,159.418
C02484=1020.994,115.627,387.781,167.528,50.857,159.419
C02485=1020.989,115.377,387.801,167.526,50.864,159.419
C02486=1020.984,115.128,387.819,167.522,50.870,159.420
C02487=1020.978,114.879,387.839,167.519,50.876,159.421
C02488=1020.973,114.630,387.858,167.517,50.882,159.421
C02489=1020.968,114.381,387.877,167.514,50.888,159.422
C02490=1020.963,114.132,387.896,167.511,50.895,159.423
C02491=1020.957,113.882,387.915,167.508,50.901,159.424
C02492=1020.952,113.634,387.934,167.505,50.906,159.424
C02493=1020.946,113.384,387.952,167.503,50.913,159.425
C02494=1020.941,113.134,387.972,167.500,50.919,159.426
C02495=1020.936,112.885,387.990,167.497,50.926,159.427
C02496=1020.930,112.636,388.010,167.494,50.931,159.427
C02497=1020.925,112.387,388.029,167.491,50.937,159.428
C02498=1020.919,112.137,388.047,167.489,50.944,159.429
C02499=1020.914,111.888,388.066,167.486,50.950,159.429
C02500=1020.909,111.639,388.085,167.482,50.957,159.430
C02501=1020.904,111.390,388.104,167.480,50.962,159.431
C02502=1020.897,111.141,388.122,167.477,50.969,159.432
C02503=1020.892,110.892,388.141,167.474,50.975,159.432
C02504=1020.887,110.642,388.160,167.471,50.982,159.433
C02505=1020.881,110.392,388.179,167.468,50.987,159.434
C02506=1020.876,110.144,388.198,167.466,50.994,159.435
C02507=1020.870,109.894,388.216,167.462,51.000,159.435
C02508=1020.865,109.645,388.234,167.460,51.007,159.436
C02509=1020.859,109.396,388.254,167.457,51.013,159.437
C02510=1020.854,109.147,388.271,167.455,51.019,159.438
C02511=1020.848,108.897,388.290,167.451,51.026,159.438
C02512=1020.843,108.648,388.309,167.448,51.032,159.439
C02513=1020.837,108.399,388.327,167.446,51.038,159.440
C02514=1020.832,108.149,388.345,167.442,51.045,159.440
C02515=1020.826,107.900,388.364,167.440,51.051,159.441
C02516=1020.820,107.617,388.385,167.437,51.058,159.442
C02517=1020.813,107.334,388.407,167.434,51.066,159.443
C02518=1020.808,107.052,388.427,167.430,51.072,159.444
C02519=1020.801,106.768,388.448,167.427,51.080,159.445
C02520=1020.796,106.519,388.467,167.424,51.086,159.445
C02521=1020.790,106.270,388.484,167.422,51.092,159.446
C02522=1020.784,106.020,388.504,167.418,51.099,159.447
C02523=1020.780,105.771,388.522,167.416,51.105,159.448
C02524=1020.773,105.522,388.540,167.414,51.112,159.448
C02525=1020.768,105.273,388.559,167.411,51.118,159.449
C02526=1020.762,105.023,388.576,167.407,51.124,159.450
C02527=1020.757,104.774,388.595,167.405,51.130,159.451
C02528=1020.752,104.525,388.614,167.402,51.137,159.451
C02529=1020.746,104.276,388.632,167.400,51.143,159.452
C02530=1020.741,104.026,388.650,167.397,51.149,159.453
C02531=1020.735,103.777,388.669,167.393,51.155,159.453
C02532=1020.730,103.528,388.687,167.391,51.162,159.454
C02533=1020.725,103.278,388.706,167.388,51.168,159.455
C02534=1020.719,103.029,388.724,167.386,51.174,159.456
C02535=1020.714,102.780,388.742,167.382,51.181,159.456
C02536=1020.708,102.531,388.761,167.380,51.187,159.457
C02537=1020.703,102.282,388.779,167.377,51.193,159.458
C02538=1020.697,102.031,388.797,167.375,51.200,159.459
C02539=1020.692,101.783,388.816,167.372,51.205,159.459
C02540=1020.687,101.534,388.834,167.369,51.212,159.460
C02541=1020.680,101.285,388.853,167.366,51.218,159.461
C02542=1020.676,101.035,388.871,167.363,51.224,159.462
C02543=1020.669,100.785,388.889,167.361,51.231,159.462
C02544=1020.664,100.537,388.908,167.358,51.237,159.463
C02545=1020.660,100.287,388.926,167.355,51.243,159.464
C02546=1020.653,100.038,388.944,167.352,51.249,159.464
C02547=1020.648,99.789,388.963,167.350,51.256,159.465
C02548=1020.643,99.540,388.980,167.347,51.262,159.466
C02549=1020.637,99.290,388.999,167.344,51.268,159.467
C02550=1020.632,99.041,389.016,167.341,51.275,159.467
C02551=1020.627,98.791,389.035,167.338,51.281,159.468
C02552=1020.621,98.542,389.053,167.336,51.287,159.469
C02553=1020.615,98.293,389.071,167.333,51.294,159.470
C02554=1020.609,98.044,389.088,167.330,51.301,159.471
C02555=1020.604,97.794,389.107,167.327,51.306,159.471
C02556=1020.599,97.545,389.124,167.325,51.313,159.472
C02557=1020.593,97.295,389.142,167.322,51.319,159.473
C02558=1020.588,97.046,389.160,167.319,51.326,159.473
C02559=1020.582,96.798,389.179,167.316,51.332,159.474
C02560=1020.576,96.548,389.197,167.314,51.338,159.475
C02561=1020.571,96.299,389.215,167.311,51.344,159.476
C02562=1020.566,96.049,389.232,167.308,51.351,159.476
C02563=1020.560,95.800,389.250,167.305,51.358,159.477
C02564=1020.554,95.551,389.268,167.303,51.364,159.478
C02565=1020.549,95.301,389.286,167.300,51.370,159.479
C02566=1020.543,95.052,389.304,167.298,51.376,159.479
C02567=1020.538,94.803,389.321,167.294,51.383,159.480
C02568=1020.533,94.553,389.340,167.291,51.389,159.481
C02569=1020.527,94.303,389.357,167.289,51.395,159.482
C02570=1020.521,94.054,389.375,167.286,51.401,159.482
C02571=1020.515,93.806,389.393,167.284,51.408,159.483
C02572=1020.511,93.557,389.412,167.280,51.414,159.484
C02573=1020.504,93.307,389.429,167.278,51.421,159.485
C02574=1020.499,93.058,389.447,167.275,51.427,159.485
C02575=1020.494,92.809,389.465,167.273,51.433,159.486
C02576=1020.489,92.560,389.483,167.270,51.439,159.487
C02577=1020.483,92.310,389.501,167.267,51.446,159.488
C02578=1020.477,92.061,389.518,167.264,51.452,159.488
C02579=1020.472,91.811,389.536,167.262,51.459,159.489
C02580=1020.465,91.528,389.556,167.259,51.466,159.490
C02581=1020.460,91.245,389.576,167.255,51.472,159.491
C02582=1020.453,90.962,389.597,167.252,51.480,159.492
C02583=1020.447,90.679,389.617,167.250,51.487,159.492
C02584=1020.442,90.430,389.635,167.246,51.493,159.493
C02585=1020.436,90.181,389.652,167.244,51.500,159.494
C02586=1020.431,89.931,389.671,167.241,51.505,159.495
C02587=1020.426,89.682,389.688,167.239,51.512,159.495
C02588=1020.420,89.433,389.706,167.236,51.518,159.496
C02589=1020.414,89.184,389.724,167.234,51.524,159.497
C02590=1020.409,88.934,389.741,167.230,51.531,159.497
C02591=1020.404,88.685,389.759,167.228,51.537,159.498
C02592=1020.398,88.436,389.776,167.225,51.543,159.499
C02593=1020.392,88.186,389.794,167.223,51.550,159.500
C02594=1020.386,87.937,389.811,167.219,51.556,159.500
C02595=1020.381,87.687,389.828,167.217,51.563,159.501
C02596=1020.375,87.438,389.846,167.214,51.569,159.502
C02597=1020.370,87.189,389.863,167.212,51.575,159.503
C02598=1020.364,86.940,389.881,167.209,51.582,159.504
C02599=1020.358,86.690,389.898,167.206,51.588,159.504
C02600=1020.353,86.441,389.915,167.204,51.595,159.505
C02601=1020.347,86.192,389.933,167.201,51.601,159.506
C02602=1020.342,85.943,389.951,167.199,51.607,159.507
C02603=1020.336,85.692,389.968,167.195,51.614,159.507
C02604=1020.331,85.443,389.985,167.193,51.620,159.508
C02605=1020.325,85.194,390.003,167.190,51.626,159.509
C02606=1020.320,84.945,390.020,167.188,51.633,159.510
C02607=1020.314,84.696,390.037,167.185,51.639,159.510
C02608=1020.309,84.447,390.055,167.182,51.646,159.511
C02609=1020.303,84.196,390.072,167.179,51.652,159.512
C02610=1020.297,83.947,390.090,167.177,51.658,159.512
C02611=1020.292,83.698,390.107,167.174,51.664,159.513
C02612=1020.287,83.448,390.124,167.172,51.671,159.514
C02613=1020.281,83.199,390.142,167.168,51.677,159.515
C02614=1020.276,82.950,390.159,167.166,51.684,159.515
C02615=1020.270,82.701,390.176,167.163,51.690,159.516
C02616=1020.264,82.451,390.194,167.161,51.696,159.517
C02617=1020.259,82.202,390.212,167.158,51.702,159.518
C02618=1020.254,81.952,390.229,167.155,51.709,159.518
C02619=1020.248,81.703,390.246,167.152,51.715,159.519
C02620=1020.242,81.455,390.263,167.150,51.722,159.520
C02621=1020.237,81.205,390.280,167.147,51.728,159.521
C02622=1020.231,80.956,390.297,167.145,51.734,159.521
C02623=1020.226,80.706,390.314,167.142,51.740,159.522
C02624=1020.220,80.457,390.332,167.140,51.746,159.523
C02625=1020.215,80.208,390.349,167.136,51.753,159.523
C02626=1020.209,79.958,390.367,167.134,51.759,159.524
C02627=1020.203,79.709,390.384,167.131,51.766,159.525
C02628=1020.198,79.459,390.401,167.129,51.772,159.526
C02629=1020.193,79.210,390.419,167.126,51.778,159.526
C02630=1020.188,78.960,390.435,167.124,51.784,159.527
C02631=1020.182,78.711,390.453,167.121,51.790,159.528
C02632=1020.177,78.462,390.471,167.118,51.797,159.529
C02633=1020.171,78.213,390.487,167.115,51.803,159.529
C02634=1020.166,77.964,390.505,167.112,51.809,159.530
C02635=1020.161,77.714,390.522,167.110,51.816,159.531
C02636=1020.155,77.465,390.539,167.108,51.822,159.531
C02637=1020.150,77.215,390.556,167.105,51.828,159.532
C02638=1020.144,76.966,390.573,167.103,51.834,159.533
C02639=1020.138,76.717,390.590,167.099,51.841,159.534
C02640=1020.133,76.467,390.607,167.097,51.847,159.534
C02641=1020.128,76.218,390.625,167.094,51.853,159.535
C02642=1020.121,75.968,390.641,167.092,51.860,159.536
C02643=1020.116,75.719,390.659,167.089,51.866,159.537
C02644=1020.109,75.436,390.678,167.086,51.874,159.538
C02645=1020.103,75.153,390.697,167.083,51.881,159.538
C02646=1020.097,74.870,390.716,167.080,51.888,159.539
C02647=1020.091,74.588,390.735,167.077,51.895,159.540
C02648=1020.085,74.338,390.751,167.074,51.901,159.541
C02649=1020.080,74.089,390.769,167.072,51.908,159.542
C02650=1020.074,73.840,390.785,167.069,51.914,159.542
C02651=1020.069,73.590,390.802,167.066,51.920,159.543
C02652=1020.063,73.341,390.820,167.063,51.927,159.544
C02653=1020.057,73.091,390.836,167.061,51.933,159.544
C02654=1020.052,72.842,390.853,167.058,51.939,159.545
C02655=1020.047,72.593,390.870,167.056,51.945,159.546
C02656=1020.041,72.343,390.887,167.054,51.952,159.547
C02657=1020.035,72.094,390.904,167.050,51.958,159.547
C02658=1020.030,71.844,390.920,167.047,51.964,159.548
C02659=1020.024,71.595,390.937,167.045,51.971,159.549
C02660=1020.019,71.346,390.954,167.042,51.977,159.549
C02661=1020.014,71.096,390.971,167.040,51.984,159.550
C02662=1020.008,70.847,390.987,167.038,51.990,159.551
C02663=1020.002,70.598,391.005,167.035,51.996,159.552
C02664=1019.996,70.348,391.021,167.032,52.003,159.552
C02665=1019.991,70.099,391.038,167.029,52.009,159.553
C02666=1019.986,69.849,391.055,167.027,52.015,159.554
C02667=1019.980,69.600,391.071,167.024,52.021,159.554
C02668=1019.974,69.351,391.089,167.022,52.028,159.555
C02669=1019.969,69.101,391.105,167.019,52.034,159.556
C02670=1019.963,68.852,391.122,167.017,52.040,159.557
C02671=1019.958,68.602,391.139,167.013,52.047,159.557
C02672=1019.952,68.353,391.155,167.011,52.053,159.558
C02673=1019.947,68.103,391.172,167.008,52.059,159.559
C02674=1019.941,67.854,391.188,167.006,52.066,159.560
C02675=1019.936,67.605,391.205,167.003,52.072,159.560
C02676=1019.930,67.356,391.221,167.001,52.078,159.561
C02677=1019.925,67.106,391.238,166.997,52.085,159.562
C02678=1019.919,66.857,391.255,166.995,52.091,159.563
C02679=1019.913,66.607,391.271,166.993,52.097,159.563
C02680=1019.908,66.358,391.288,166.990,52.103,159.564
C02681=1019.902,66.108,391.304,166.988,52.110,159.565
C02682=1019.896,65.859,391.321,166.985,52.116,159.565
C02683=1019.891,65.609,391.338,166.982,52.123,159.566
C02684=1019.885,65.360,391.354,166.979,52.129,159.567
C02685=1019.880,65.111,391.370,166.977,52.135,159.567
C02686=1019.875,64.862,391.387,166.974,52.142,159.568
C02687=1019.869,64.612,391.403,166.972,52.148,159.569
C02688=1019.863,64.363,391.420,166.970,52.154,159.570
C02689=1019.858,64.113,391.436,166.966,52.161,159.570
C02690=1019.852,63.864,391.453,166.963,52.167,159.571
C02691=1019.846,63.614,391.469,166.961,52.173,159.572
C02692=1019.840,63.365,391.485,166.958,52.179,159.573
C02693=1019.836,63.116,391.502,166.956,52.185,159.573
C02694=1019.830,62.867,391.518,166.954,52.192,159.574
C02695=1019.824,62.617,391.534,166.950,52.198,159.575
C02696=1019.818,62.367,391.550,166.948,52.205,159.576
C02697=1019.813,62.118,391.567,166.946,52.212,159.576
C02698=1019.807,61.868,391.583,166.943,52.218,159.577
C02699=1019.801,61.619,391.599,166.940,52.225,159.578
C02700=1019.796,61.369,391.615,166.937,52.231,159.578
C02701=1019.790,61.120,391.631,166.935,52.237,159.579
C02702=1019.784,60.871,391.647,166.932,52.243,159.580
C02703=1019.778,60.622,391.663,166.930,52.250,159.581
C02704=1019.772,60.372,391.679,166.926,52.257,159.581
C02705=1019.767,60.122,391.695,166.924,52.263,159.582
C02706=1019.761,59.873,391.712,166.922,52.269,159.583
C02707=1019.756,59.624,391.728,166.919,52.276,159.584
C02708=1019.749,59.341,391.745,166.916,52.283,159.585
C02709=1019.743,59.058,391.764,166.913,52.290,159.585
C02710=1019.737,58.775,391.782,166.910,52.298,159.586
C02711=1019.730,58.492,391.800,166.907,52.305,159.587
C02712=1019.725,58.242,391.817,166.904,52.311,159.588
C02713=1019.719,57.993,391.833,166.902,52.318,159.589
C02714=1019.713,57.743,391.849,166.899,52.324,159.589
C02715=1019.708,57.494,391.864,166.896,52.331,159.590
C02716=1019.702,57.245,391.880,166.894,52.337,159.591
C02717=1019.696,56.995,391.897,166.892,52.343,159.591
C02718=1019.690,56.745,391.912,166.889,52.350,159.592
C02719=1019.684,56.496,391.929,166.885,52.356,159.593
C02720=1019.679,56.247,391.944,166.883,52.363,159.594
C02721=1019.673,55.997,391.960,166.881,52.369,159.594
C02722=1019.668,55.748,391.977,166.879,52.375,159.595
C02723=1019.662,55.498,391.993,166.876,52.381,159.596
C02724=1019.657,55.249,392.008,166.872,52.388,159.596
C02725=1019.651,55.000,392.024,166.870,52.394,159.597
C02726=1019.645,54.750,392.041,166.868,52.400,159.598
C02727=1019.640,54.500,392.056,166.865,52.406,159.598
C02728=1019.634,54.252,392.072,166.863,52.413,159.599
C02729=1019.629,54.002,392.088,166.860,52.419,159.600
C02730=1019.623,53.752,392.104,166.858,52.425,159.601
C02731=1019.617,53.504,392.120,166.854,52.432,159.601
C02732=1019.612,53.254,392.135,166.852,52.438,159.602
C02733=1019.606,53.004,392.152,166.849,52.444,159.603
C02734=1019.601,52.754,392.168,166.847,52.451,159.604
C02735=1019.595,52.506,392.184,166.845,52.457,159.604
C02736=1019.589,52.256,392.200,166.842,52.463,159.605
C02737=1019.584,52.006,392.215,166.839,52.470,159.606
C02738=1019.578,51.758,392.231,166.836,52.476,159.606
C02739=1019.573,51.508,392.247,166.834,52.482,159.607
C02740=1019.567,51.258,392.263,166.831,52.489,159.608
C02741=1019.562,51.009,392.278,166.829,52.495,159.608
C02742=1019.556,50.760,392.295,166.826,52.501,159.609
C02743=1019.550,50.510,392.310,166.824,52.507,159.610
C02744=1019.546,50.261,392.327,166.822,52.514,159.611
C02745=1019.540,50.011,392.342,166.818,52.520,159.611
C02746=1019.534,49.761,392.358,166.815,52.526,159.612
C02747=1019.529,49.512,392.374,166.813,52.532,159.612
C02748=1019.523,49.263,392.390,166.811,52.539,159.613
C02749=1019.517,49.013,392.405,166.808,52.545,159.614
C02750=1019.512,48.764,392.421,166.805,52.551,159.615
C02751=1019.506,48.514,392.437,166.803,52.557,159.615
C02752=1019.500,48.265,392.453,166.800,52.563,159.616
C02753=1019.495,48.016,392.468,166.798,52.570,159.617
C02754=1019.489,47.766,392.485,166.795,52.576,159.617
C02755=1019.484,47.517,392.500,166.792,52.582,159.618
C02756=1019.478,47.268,392.516,166.789,52.589,159.619
C02757=1019.474,47.017,392.532,166.787,52.595,159.619
C02758=1019.468,46.769,392.548,166.784,52.601,159.620
C02759=1019.463,46.519,392.564,166.782,52.607,159.621
C02760=1019.457,46.269,392.579,166.780,52.613,159.622
C02761=1019.452,46.020,392.595,166.777,52.619,159.622
C02762=1019.446,45.770,392.610,166.775,52.626,159.623
C02763=1019.441,45.522,392.626,166.772,52.632,159.624
C02764=1019.435,45.272,392.642,166.769,52.638,159.624
C02765=1019.430,45.022,392.657,166.767,52.644,159.625
C02766=1019.424,44.773,392.673,166.764,52.651,159.626
C02767=1019.419,44.524,392.689,166.761,52.657,159.626
C02768=1019.413,44.274,392.705,166.759,52.663,159.627
C02769=1019.407,44.024,392.720,166.756,52.669,159.628
C02770=1019.402,43.775,392.735,166.753,52.675,159.628
C02771=1019.397,43.525,392.752,166.751,52.681,159.629
C02772=1019.391,43.243,392.770,166.748,52.688,159.630
C02773=1019.384,42.960,392.787,166.746,52.695,159.630
C02774=1019.378,42.676,392.806,166.742,52.702,159.631
C02775=1019.372,42.393,392.822,166.739,52.709,159.632
C02776=1019.367,42.144,392.838,166.737,52.715,159.633
C02777=1019.361,41.894,392.854,166.734,52.721,159.633
C02778=1019.356,41.645,392.869,166.732,52.728,159.634
C02779=1019.350,41.395,392.884,166.730,52.734,159.635
C02780=1019.345,41.146,392.899,166.726,52.741,159.635
C02781=1019.339,40.896,392.915,166.723,52.747,159.636
C02782=1019.334,40.647,392.931,166.721,52.753,159.637
C02783=1019.327,40.397,392.946,166.719,52.759,159.638
C02784=1019.322,40.148,392.961,166.716,52.766,159.638
C02785=1019.317,39.898,392.976,166.714,52.772,159.639
C02786=1019.311,39.649,392.991,166.711,52.778,159.639
C02787=1019.306,39.399,393.007,166.708,52.784,159.640
C02788=1019.300,39.151,393.022,166.705,52.791,159.641
C02789=1019.294,38.901,393.038,166.703,52.797,159.642
C02790=1019.289,38.651,393.053,166.700,52.803,159.642
C02791=1019.283,38.401,393.069,166.698,52.809,159.643
C02792=1019.278,38.152,393.083,166.695,52.815,159.644
C02793=1019.272,37.903,393.099,166.693,52.822,159.644
C02794=1019.267,37.653,393.114,166.691,52.828,159.645
C02795=1019.261,37.403,393.129,166.687,52.834,159.646
C02796=1019.256,37.154,393.145,166.684,52.841,159.646
C02797=1019.250,36.904,393.160,166.682,52.847,159.647
C02798=1019.245,36.655,393.175,166.679,52.853,159.648
C02799=1019.239,36.405,393.190,166.677,52.859,159.648
C02800=1019.233,36.156,393.205,166.675,52.866,159.649
C02801=1019.228,35.906,393.220,166.671,52.872,159.650
C02802=1019.222,35.657,393.235,166.669,52.878,159.650
C02803=1019.216,35.407,393.250,166.667,52.885,159.651
C02804=1019.211,35.158,393.265,166.664,52.891,159.652
C02805=1019.205,34.908,393.281,166.662,52.897,159.652
C02806=1019.200,34.659,393.296,166.658,52.903,159.653
C02807=1019.194,34.410,393.310,166.656,52.910,159.654
C02808=1019.188,34.160,393.326,166.653,52.916,159.655
C02809=1019.183,33.911,393.340,166.651,52.922,159.655
C02810=1019.177,33.661,393.356,166.648,52.928,159.656
C02811=1019.172,33.412,393.370,166.646,52.935,159.657
C02812=1019.166,33.162,393.385,166.643,52.942,159.657
C02813=1019.160,32.913,393.400,166.640,52.948,159.658
C02814=1019.155,32.663,393.415,166.638,52.954,159.659
C02815=1019.149,32.414,393.430,166.635,52.960,159.659
C02816=1019.144,32.165,393.445,166.633,52.967,159.660
C02817=1019.137,31.915,393.460,166.629,52.973,159.661
C02818=1019.133,31.665,393.475,166.627,52.979,159.661
C02819=1019.127,31.416,393.489,166.624,52.985,159.662
C02820=1019.121,31.166,393.505,166.622,52.992,159.663
C02821=1019.115,30.917,393.519,166.619,52.998,159.663
C02822=1019.110,30.667,393.535,166.617,53.004,159.664
C02823=1019.104,30.418,393.550,166.614,53.011,159.665
C02824=1019.099,30.168,393.564,166.611,53.017,159.665
C02825=1019.093,29.919,393.579,166.609,53.023,159.666
C02826=1019.088,29.669,393.594,166.606,53.029,159.667
C02827=1019.082,29.420,393.609,166.604,53.035,159.667
C02828=1019.076,29.170,393.624,166.601,53.041,159.668
C02829=1019.071,28.921,393.638,166.599,53.048,159.669
C02830=1019.066,28.672,393.653,166.596,53.055,159.669
C02831=1019.059,28.422,393.668,166.593,53.061,159.670
C02832=1019.054,28.173,393.683,166.591,53.067,159.671
C02833=1019.050,27.923,393.698,166.588,53.073,159.671
C02834=1019.043,27.673,393.713,166.586,53.079,159.672
C02835=1019.037,27.424,393.727,166.583,53.085,159.673
C02836=1019.031,27.140,393.744,166.580,53.092,159.673
C02837=1019.025,26.857,393.761,166.577,53.100,159.674
C02838=1019.018,26.574,393.777,166.574,53.107,159.675
C02839=1019.013,26.291,393.794,166.571,53.114,159.676
C02840=1019.007,26.042,393.808,166.569,53.121,159.676
C02841=1019.001,25.792,393.824,166.566,53.127,159.677
C02842=1018.996,25.542,393.838,166.563,53.133,159.678
C02843=1018.990,25.293,393.852,166.560,53.139,159.678
C02844=1018.984,25.043,393.867,166.558,53.146,159.679
C02845=1018.979,24.794,393.882,166.555,53.152,159.680
C02846=1018.973,24.544,393.896,166.553,53.158,159.680
C02847=1018.967,24.295,393.910,166.550,53.165,159.681
C02848=1018.961,24.046,393.925,166.547,53.171,159.682
C02849=1018.956,23.796,393.940,166.545,53.177,159.682
C02850=1018.951,23.547,393.954,166.542,53.183,159.683
C02851=1018.945,23.296,393.968,166.540,53.190,159.684
C02852=1018.939,23.047,393.984,166.536,53.197,159.684
C02853=1018.934,22.798,393.998,166.534,53.203,159.685
C02854=1018.928,22.549,394.012,166.532,53.209,159.686
C02855=1018.922,22.298,394.026,166.529,53.215,159.686
C02856=1018.917,22.049,394.041,166.527,53.221,159.687
C02857=1018.912,21.800,394.055,166.523,53.228,159.687
C02858=1018.906,21.551,394.070,166.521,53.234,159.688
C02859=1018.900,21.301,394.084,166.518,53.241,159.689
C02860=1018.895,21.051,394.099,166.516,53.247,159.690
C02861=1018.889,20.802,394.113,166.514,53.253,159.690
C02862=1018.883,20.553,394.128,166.510,53.259,159.691
C02863=1018.878,20.303,394.142,166.508,53.265,159.691
C02864=1018.873,20.052,394.156,166.505,53.272,159.692
C02865=1018.867,19.803,394.171,166.503,53.278,159.693
C02866=1018.861,19.554,394.185,166.500,53.284,159.693
C02867=1018.856,19.305,394.200,166.498,53.290,159.694
C02868=1018.851,19.055,394.214,166.494,53.296,159.695
C02869=1018.844,18.805,394.229,166.492,53.303,159.695
C02870=1018.839,18.556,394.243,166.490,53.309,159.696
C02871=1018.834,18.306,394.257,166.487,53.316,159.697
C02872=1018.828,18.057,394.271,166.484,53.322,159.697
C02873=1018.822,17.808,394.285,166.481,53.328,159.698
C02874=1018.817,17.558,394.299,166.479,53.334,159.699
C02875=1018.811,17.308,394.313,166.476,53.340,159.699
C02876=1018.806,17.059,394.328,166.474,53.347,159.700
C02877=1018.800,16.809,394.342,166.470,53.353,159.700
C02878=1018.795,16.559,394.356,166.468,53.360,159.701
C02879=1018.789,16.310,394.371,166.466,53.366,159.702
C02880=1018.783,16.061,394.385,166.463,53.372,159.703
C02881=1018.777,15.811,394.399,166.461,53.378,159.703
C02882=1018.772,15.562,394.413,166.457,53.385,159.704
C02883=1018.766,15.312,394.427,166.455,53.391,159.704
C02884=1018.761,15.062,394.441,166.452,53.397,159.705
C02885=1018.755,14.813,394.455,166.450,53.403,159.706
C02886=1018.750,14.564,394.470,166.446,53.410,159.706
C02887=1018.745,14.314,394.484,166.444,53.416,159.707
C02888=1018.739,14.065,394.498,166.441,53.422,159.708
C02889=1018.733,13.814,394.512,166.439,53.428,159.708
C02890=1018.728,13.565,394.526,166.437,53.434,159.709
C02891=1018.722,13.316,394.541,166.434,53.441,159.710
C02892=1018.716,13.066,394.554,166.431,53.448,159.710
C02893=1018.711,12.817,394.568,166.429,53.454,159.711
C02894=1018.705,12.567,394.582,166.426,53.460,159.712
C02895=1018.699,12.318,394.595,166.423,53.467,159.712
C02896=1018.694,12.068,394.609,166.420,53.473,159.713
C02897=1018.688,11.819,394.623,166.418,53.480,159.714
C02898=1018.683,11.569,394.637,166.415,53.486,159.714
C02899=1018.677,11.319,394.651,166.412,53.492,159.715
C02900=1018.671,11.090,394.664,166.410,53.498,159.715
C02901=1018.666,10.860,394.676,166.407,53.504,159.716
C02902=1018.661,10.629,394.689,166.404,53.510,159.717
C02903=1018.656,10.400,394.702,166.403,53.516,159.717
C02904=1018.650,10.169,394.714,166.400,53.521,159.718
C02905=1018.645,9.940,394.727,166.398,53.527,159.718
C02906=1018.641,9.710,394.740,166.395,53.534,159.719
C02907=1018.635,9.480,394.753,166.392,53.539,159.720
C02908=1018.629,9.231,394.767,166.390,53.546,159.720
C02909=1018.624,8.981,394.781,166.388,53.552,159.721
C02910=1018.618,8.732,394.794,166.384,53.559,159.722
C02911=1018.612,8.482,394.808,166.382,53.565,159.722
C02912=1018.607,8.232,394.821,166.379,53.571,159.723
C02913=1018.601,7.982,394.835,166.376,53.577,159.723
C02914=1018.596,7.733,394.849,166.374,53.584,159.724
C02915=1018.590,7.484,394.862,166.371,53.590,159.725
C02916=1018.584,7.234,394.876,166.369,53.596,159.725
C02917=1018.579,6.984,394.890,166.365,53.602,159.726
C02918=1018.573,6.735,394.903,166.363,53.609,159.727
C02919=1018.568,6.485,394.917,166.361,53.616,159.727
C02920=1018.562,6.236,394.931,166.358,53.622,159.728
C02921=1018.556,5.986,394.944,166.355,53.628,159.729
C02922=1018.551,5.737,394.958,166.352,53.634,159.729
C02923=1018.545,5.487,394.972,166.350,53.641,159.730
C02924=1018.540,5.237,394.985,166.346,53.647,159.730
C02925=1018.534,4.988,394.999,166.344,53.653,159.731
C02926=1018.528,4.738,395.012,166.342,53.659,159.732
C02927=1018.523,4.489,395.026,166.339,53.666,159.732
C02928=1018.517,4.239,395.040,166.336,53.672,159.733
C02929=1018.512,3.990,395.054,166.333,53.678,159.733
C02930=1018.506,3.740,395.067,166.331,53.685,159.734
C02931=1018.501,3.490,395.081,166.328,53.691,159.735
C02932=1018.495,3.240,395.094,166.325,53.697,159.735
C02933=1018.490,2.992,395.108,166.323,53.703,159.736
C02934=1018.485,2.742,395.122,166.320,53.710,159.737
C02935=1018.479,2.493,395.135,166.318,53.716,159.737
C02936=1018.473,2.243,395.149,166.315,53.722,159.738
C02937=1018.468,1.993,395.162,166.312,53.729,159.738
C02938=1018.462,1.743,395.176,166.309,53.735,159.739
C02939=1018.456,1.494,395.189,166.307,53.741,159.740
C02940=1018.451,1.245,395.203,166.305,53.747,159.740
C02941=1018.446,0.994,395.216,166.301,53.754,159.741
C02942=1018.440,0.745,395.230,166.299,53.760,159.742
C02943=1018.435,0.495,395.244,166.296,53.765,159.742
C02944=1018.427,0.174,395.261,166.292,53.774,159.743
C02945=1018.421,-0.147,395.278,166.289,53.782,159.744
C02946=1018.413,-0.468,395.295,166.286,53.789,159.744
C02947=1018.407,-0.788,395.314,166.282,53.798,159.745
C02948=1018.401,-1.038,395.326,166.280,53.804,159.746
C02949=1018.395,-1.288,395.340,166.277,53.810,159.746
C02950=1018.390,-1.537,395.353,166.273,53.816,159.747
C02951=1018.385,-1.787,395.367,166.271,53.822,159.747
C02952=1018.379,-2.036,395.380,166.268,53.828,159.748
C02953=1018.373,-2.286,395.394,166.266,53.835,159.749
C02954=1018.368,-2.535,395.408,166.264,53.841,159.749
C02955=1018.363,-2.786,395.421,166.260,53.847,159.750
C02956=1018.358,-3.034,395.434,166.258,53.854,159.751
C02957=1018.352,-3.284,395.448,166.255,53.859,159.751
C02958=1018.347,-3.534,395.461,166.253,53.865,159.752
C02959=1018.341,-3.783,395.475,166.250,53.871,159.752
C02960=1018.336,-4.034,395.488,166.247,53.878,159.753
C02961=1018.330,-4.283,395.501,166.244,53.884,159.753
C02962=1018.325,-4.532,395.514,166.242,53.890,159.754
C02963=1018.319,-4.782,395.527,166.239,53.897,159.755
C02964=1018.313,-5.061,395.542,166.237,53.904,159.755
C02965=1018.306,-5.341,395.557,166.233,53.910,159.756
C02966=1018.300,-5.621,395.571,166.230,53.918,159.757
C02967=1018.294,-5.901,395.585,166.227,53.925,159.757
C02968=1018.288,-6.150,395.599,166.224,53.932,159.758
C02969=1018.283,-6.401,395.612,166.221,53.938,159.759
C02970=1018.277,-6.649,395.625,166.219,53.944,159.759
C02971=1018.271,-6.899,395.637,166.215,53.951,159.760
C02972=1018.266,-7.149,395.651,166.213,53.957,159.760
C02973=1018.260,-7.398,395.664,166.211,53.963,159.761
C02974=1018.255,-7.649,395.677,166.207,53.970,159.762
C02975=1018.249,-7.897,395.690,166.205,53.976,159.762
C02976=1018.244,-8.147,395.703,166.202,53.982,159.763
C02977=1018.238,-8.397,395.716,166.199,53.989,159.763
C02978=1018.232,-8.647,395.729,166.197,53.995,159.764
C02979=1018.227,-8.896,395.742,166.194,54.001,159.765
C02980=1018.221,-9.146,395.754,166.191,54.008,159.765
C02981=1018.216,-9.396,395.768,166.188,54.014,159.766
C02982=1018.211,-9.645,395.780,166.186,54.020,159.766
C02983=1018.205,-9.895,395.793,166.183,54.027,159.767
C02984=1018.199,-10.144,395.807,166.180,54.033,159.768
C02985=1018.193,-10.394,395.819,166.178,54.039,159.768
C02986=1018.189,-10.644,395.832,166.174,54.046,159.769
C02987=1018.182,-10.893,395.845,166.172,54.051,159.769
C02988=1018.177,-11.143,395.858,166.169,54.057,159.770
C02989=1018.172,-11.392,395.871,166.166,54.064,159.770
C02990=1018.166,-11.642,395.883,166.163,54.070,159.771
C02991=1018.161,-11.892,395.897,166.161,54.077,159.772
C02992=1018.155,-12.141,395.909,166.159,54.083,159.772
C02993=1018.149,-12.391,395.922,166.155,54.089,159.773
C02994=1018.144,-12.641,395.935,166.153,54.096,159.773
C02995=1018.139,-12.889,395.948,166.150,54.102,159.774
C02996=1018.133,-13.139,395.960,166.146,54.108,159.774
C02997=1018.128,-13.390,395.973,166.144,54.114,159.775
C02998=1018.122,-13.639,395.986,166.142,54.120,159.776
C02999=1018.117,-13.888,396.000,166.139,54.126,159.776
C03000=1018.111,-14.137,396.012,166.136,54.133,159.777
C03001=1018.106,-14.387,396.024,166.134,54.139,159.777
C03002=1018.100,-14.638,396.037,166.131,54.145,159.778
C03003=1018.095,-14.887,396.050,166.127,54.151,159.778
C03004=1018.090,-15.136,396.063,166.125,54.158,159.779
C03005=1018.084,-15.386,396.076,166.123,54.164,159.780
C03006=1018.078,-15.635,396.088,166.120,54.170,159.780
C03007=1018.073,-15.886,396.101,166.117,54.177,159.781
C03008=1018.068,-16.135,396.114,166.114,54.182,159.781
C03009=1018.062,-16.385,396.126,166.112,54.188,159.782
C03010=1018.056,-16.635,396.139,166.108,54.195,159.782
C03011=1018.051,-16.884,396.151,166.106,54.201,159.783
C03012=1018.045,-17.134,396.163,166.102,54.208,159.784
C03013=1018.040,-17.383,396.176,166.100,54.214,159.784
C03014=1018.034,-17.633,396.189,166.098,54.220,159.785
C03015=1018.029,-17.882,396.201,166.094,54.227,159.785
C03016=1018.023,-18.132,396.213,166.092,54.233,159.786
C03017=1018.017,-18.382,396.226,166.090,54.239,159.787
C03018=1018.012,-18.631,396.238,166.086,54.246,159.787
C03019=1018.006,-18.881,396.251,166.084,54.252,159.788
C03020=1018.001,-19.130,396.263,166.080,54.259,159.788
C03021=1017.995,-19.380,396.276,166.078,54.265,159.789
C03022=1017.990,-19.630,396.288,166.076,54.271,159.790
C03023=1017.984,-19.879,396.301,166.072,54.278,159.790
C03024=1017.979,-20.129,396.313,166.070,54.284,159.791
C03025=1017.973,-20.378,396.326,166.067,54.290,159.791
C03026=1017.968,-20.628,396.338,166.064,54.297,159.792
C03027=1017.962,-20.878,396.350,166.061,54.303,159.792
C03028=1017.957,-21.156,396.364,166.058,54.310,159.793
C03029=1017.950,-21.434,396.377,166.055,54.317,159.794
C03030=1017.943,-21.712,396.392,166.052,54.324,159.794
C03031=1017.938,-21.990,396.405,166.049,54.331,159.795
C03032=1017.932,-22.239,396.418,166.046,54.337,159.795
C03033=1017.927,-22.489,396.430,166.043,54.344,159.796
C03034=1017.922,-22.738,396.442,166.041,54.350,159.797
C03035=1017.916,-22.988,396.454,166.038,54.356,159.797
C03036=1017.910,-23.237,396.466,166.034,54.362,159.797
C03037=1017.905,-23.487,396.479,166.032,54.368,159.798
C03038=1017.899,-23.737,396.491,166.030,54.375,159.799
C03039=1017.894,-23.987,396.504,166.026,54.381,159.799
C03040=1017.889,-24.237,396.516,166.024,54.387,159.800
C03041=1017.883,-24.486,396.528,166.021,54.393,159.800
C03042=1017.878,-24.736,396.540,166.018,54.400,159.801
C03043=1017.872,-24.985,396.553,166.015,54.406,159.802
C03044=1017.867,-25.235,396.565,166.013,54.412,159.802
C03045=1017.862,-25.484,396.577,166.010,54.419,159.803
C03046=1017.856,-25.734,396.589,166.007,54.424,159.803
C03047=1017.850,-25.983,396.601,166.005,54.431,159.804
C03048=1017.844,-26.233,396.614,166.001,54.437,159.804
C03049=1017.839,-26.483,396.625,165.999,54.444,159.805
C03050=1017.835,-26.733,396.638,165.996,54.449,159.805
C03051=1017.829,-26.983,396.651,165.993,54.456,159.806
C03052=1017.824,-27.232,396.663,165.990,54.462,159.806
C03053=1017.818,-27.482,396.675,165.988,54.468,159.807
C03054=1017.813,-27.731,396.687,165.984,54.474,159.807
C03055=1017.807,-27.982,396.699,165.982,54.481,159.808
C03056=1017.802,-28.231,396.711,165.979,54.487,159.809
C03057=1017.796,-28.480,396.723,165.976,54.493,159.809
C03058=1017.790,-28.730,396.734,165.974,54.500,159.810
C03059=1017.785,-28.980,396.747,165.970,54.506,159.810
C03060=1017.780,-29.229,396.758,165.968,54.513,159.811
C03061=1017.774,-29.479,396.771,165.964,54.519,159.811
C03062=1017.768,-29.729,396.781,165.962,54.525,159.812
C03063=1017.763,-29.978,396.794,165.960,54.531,159.812
C03064=1017.757,-30.229,396.805,165.956,54.538,159.813
C03065=1017.752,-30.478,396.818,165.954,54.544,159.814
C03066=1017.747,-30.728,396.829,165.951,54.551,159.814
C03067=1017.740,-30.977,396.841,165.948,54.557,159.815
C03068=1017.735,-31.227,396.853,165.945,54.563,159.815
C03069=1017.730,-31.476,396.865,165.942,54.569,159.816
C03070=1017.725,-31.727,396.877,165.940,54.576,159.816
C03071=1017.719,-31.976,396.889,165.936,54.582,159.817
C03072=1017.713,-32.225,396.900,165.934,54.588,159.817
C03073=1017.708,-32.475,396.912,165.930,54.594,159.818
C03074=1017.703,-32.725,396.924,165.928,54.601,159.818
C03075=1017.697,-32.974,396.936,165.926,54.607,159.819
C03076=1017.692,-33.224,396.947,165.922,54.614,159.819
C03077=1017.686,-33.473,396.959,165.920,54.620,159.820
C03078=1017.681,-33.723,396.971,165.917,54.626,159.821
C03079=1017.676,-33.973,396.982,165.914,54.632,159.821
C03080=1017.670,-34.223,396.995,165.911,54.639,159.822
C03081=1017.665,-34.473,397.006,165.908,54.645,159.822
C03082=1017.659,-34.722,397.018,165.905,54.651,159.823
C03083=1017.654,-34.971,397.029,165.903,54.657,159.823
C03084=1017.649,-35.221,397.041,165.900,54.664,159.824
C03085=1017.643,-35.471,397.053,165.897,54.670,159.824
C03086=1017.638,-35.721,397.065,165.893,54.676,159.825
C03087=1017.632,-35.970,397.076,165.891,54.682,159.825
C03088=1017.627,-36.220,397.088,165.889,54.689,159.826
C03089=1017.621,-36.470,397.100,165.885,54.695,159.826
C03090=1017.616,-36.719,397.112,165.883,54.701,159.827
C03091=1017.611,-36.969,397.123,165.880,54.707,159.827
C03092=1017.604,-37.246,397.136,165.877,54.714,159.828
C03093=1017.599,-37.523,397.149,165.874,54.721,159.829
C03094=1017.592,-37.800,397.162,165.871,54.728,159.829
C03095=1017.587,-38.077,397.175,165.867,54.735,159.830
C03096=1017.581,-38.327,397.186,165.864,54.741,159.830
C03097=1017.576,-38.577,397.197,165.861,54.747,159.831
C03098=1017.570,-38.826,397.210,165.859,54.753,159.831
C03099=1017.565,-39.076,397.221,165.856,54.760,159.832
C03100=1017.560,-39.326,397.232,165.853,54.765,159.832
C03101=1017.555,-39.576,397.244,165.851,54.772,159.833
C03102=1017.550,-39.825,397.255,165.847,54.778,159.833
C03103=1017.543,-40.074,397.267,165.845,54.785,159.834
C03104=1017.538,-40.325,397.279,165.842,54.791,159.834
C03105=1017.532,-40.574,397.290,165.839,54.797,159.835
C03106=1017.527,-40.824,397.301,165.836,54.804,159.835
C03107=1017.521,-41.073,397.312,165.833,54.810,159.836
C03108=1017.516,-41.323,397.323,165.830,54.817,159.836
C03109=1017.511,-41.573,397.334,165.828,54.823,159.837
C03110=1017.506,-41.823,397.346,165.824,54.829,159.837
C03111=1017.500,-42.072,397.357,165.821,54.835,159.838
C03112=1017.495,-42.322,397.368,165.819,54.842,159.839
C03113=1017.489,-42.572,397.379,165.816,54.848,159.839
C03114=1017.484,-42.822,397.391,165.813,54.854,159.839
C03115=1017.478,-43.071,397.402,165.810,54.861,159.840
C03116=1017.473,-43.321,397.413,165.807,54.867,159.841
C03117=1017.467,-43.570,397.425,165.804,54.874,159.841
C03118=1017.462,-43.820,397.436,165.801,54.879,159.841
C03119=1017.456,-44.069,397.447,165.799,54.886,159.842
C03120=1017.451,-44.319,397.459,165.796,54.892,159.843
C03121=1017.445,-44.569,397.469,165.793,54.898,159.843
C03122=1017.440,-44.818,397.481,165.790,54.905,159.843
C03123=1017.435,-45.068,397.492,165.787,54.911,159.844
C03124=1017.430,-45.318,397.503,165.784,54.918,159.845
C03125=1017.424,-45.568,397.513,165.781,54.923,159.845
C03126=1017.419,-45.818,397.525,165.779,54.930,159.846
C03127=1017.413,-46.067,397.536,165.776,54.936,159.846
C03128=1017.408,-46.317,397.547,165.773,54.942,159.847
C03129=1017.403,-46.566,397.558,165.770,54.949,159.847
C03130=1017.398,-46.816,397.570,165.767,54.955,159.848
C03131=1017.392,-47.066,397.581,165.764,54.961,159.848
C03132=1017.387,-47.315,397.592,165.761,54.967,159.849
C03133=1017.381,-47.565,397.603,165.759,54.974,159.849
C03134=1017.376,-47.815,397.614,165.755,54.980,159.849
C03135=1017.370,-48.064,397.625,165.753,54.986,159.850
C03136=1017.365,-48.314,397.637,165.749,54.992,159.850
C03137=1017.360,-48.564,397.647,165.747,54.998,159.851
C03138=1017.355,-48.814,397.658,165.745,55.005,159.852
C03139=1017.349,-49.063,397.669,165.741,55.011,159.852
C03140=1017.344,-49.313,397.681,165.738,55.017,159.853
C03141=1017.338,-49.563,397.692,165.735,55.023,159.853
C03142=1017.333,-49.813,397.703,165.732,55.029,159.853
C03143=1017.328,-50.062,397.714,165.730,55.035,159.854
C03144=1017.323,-50.312,397.725,165.726,55.042,159.854
C03145=1017.317,-50.562,397.736,165.724,55.048,159.855
C03146=1017.312,-50.812,397.747,165.721,55.053,159.855
C03147=1017.307,-51.061,397.758,165.718,55.060,159.856
C03148=1017.301,-51.311,397.769,165.716,55.067,159.856
C03149=1017.295,-51.561,397.779,165.712,55.073,159.857
C03150=1017.290,-51.810,397.790,165.710,55.079,159.857
C03151=1017.285,-52.060,397.800,165.706,55.086,159.858
C03152=1017.280,-52.310,397.811,165.703,55.092,159.858
C03153=1017.274,-52.560,397.821,165.701,55.099,159.859
C03154=1017.269,-52.809,397.832,165.697,55.105,159.859
C03155=1017.263,-53.059,397.843,165.695,55.111,159.860
C03156=1017.257,-53.336,397.854,165.692,55.119,159.861
C03157=1017.251,-53.614,397.866,165.688,55.126,159.861
C03158=1017.245,-53.891,397.878,165.685,55.133,159.862
C03159=1017.239,-54.168,397.890,165.681,55.140,159.862
C03160=1017.233,-54.418,397.900,165.679,55.146,159.863
C03161=1017.227,-54.667,397.911,165.676,55.153,159.863
C03162=1017.222,-54.917,397.921,165.674,55.159,159.864
C03163=1017.216,-55.167,397.932,165.670,55.165,159.864
C03164=1017.211,-55.416,397.942,165.668,55.172,159.865
C03165=1017.206,-55.666,397.952,165.664,55.178,159.865
C03166=1017.201,-55.916,397.963,165.661,55.185,159.866
C03167=1017.195,-56.166,397.974,165.658,55.191,159.866
C03168=1017.190,-56.416,397.984,165.655,55.198,159.867
C03169=1017.184,-56.665,397.995,165.653,55.204,159.867
C03170=1017.179,-56.915,398.005,165.649,55.210,159.867
C03171=1017.174,-57.165,398.015,165.647,55.216,159.868
C03172=1017.168,-57.414,398.026,165.643,55.223,159.869
C03173=1017.163,-57.664,398.036,165.641,55.229,159.869
C03174=1017.157,-57.914,398.047,165.637,55.235,159.869
C03175=1017.152,-58.163,398.057,165.635,55.242,159.870
C03176=1017.146,-58.413,398.068,165.632,55.249,159.871
C03177=1017.141,-58.663,398.078,165.629,55.254,159.871
C03178=1017.136,-58.913,398.088,165.626,55.261,159.871
C03179=1017.130,-59.162,398.098,165.624,55.267,159.872
C03180=1017.125,-59.412,398.109,165.620,55.273,159.872
C03181=1017.120,-59.662,398.120,165.618,55.280,159.873
C03182=1017.115,-59.912,398.130,165.614,55.286,159.873
C03183=1017.110,-60.161,398.140,165.612,55.292,159.874
C03184=1017.104,-60.411,398.151,165.608,55.299,159.874
C03185=1017.099,-60.661,398.161,165.606,55.305,159.875
C03186=1017.093,-60.911,398.171,165.603,55.311,159.875
C03187=1017.088,-61.160,398.182,165.600,55.318,159.876
C03188=1017.083,-61.410,398.192,165.597,55.323,159.876
C03189=1017.077,-61.660,398.202,165.594,55.330,159.877
C03190=1017.072,-61.909,398.213,165.591,55.336,159.877
C03191=1017.066,-62.159,398.223,165.588,55.342,159.878
C03192=1017.061,-62.409,398.233,165.586,55.349,159.878
C03193=1017.056,-62.659,398.243,165.582,55.355,159.878
C03194=1017.050,-62.908,398.254,165.580,55.361,159.879
C03195=1017.045,-63.158,398.264,165.576,55.367,159.879
C03196=1017.040,-63.408,398.274,165.574,55.374,159.880
C03197=1017.035,-63.657,398.284,165.570,55.380,159.880
C03198=1017.029,-63.907,398.295,165.568,55.386,159.881
C03199=1017.024,-64.157,398.305,165.565,55.392,159.881
C03200=1017.020,-64.407,398.315,165.562,55.399,159.882
C03201=1017.014,-64.657,398.325,165.560,55.405,159.882
C03202=1017.009,-64.906,398.336,165.556,55.411,159.883
C03203=1017.004,-65.156,398.346,165.554,55.417,159.883
C03204=1016.998,-65.406,398.356,165.550,55.423,159.883
C03205=1016.993,-65.655,398.366,165.548,55.430,159.884
C03206=1016.988,-65.905,398.376,165.545,55.435,159.884
C03207=1016.982,-66.155,398.387,165.542,55.442,159.885
C03208=1016.977,-66.404,398.397,165.539,55.448,159.885
C03209=1016.972,-66.654,398.407,165.535,55.454,159.885
C03210=1016.967,-66.904,398.417,165.533,55.460,159.886
C03211=1016.962,-67.154,398.427,165.529,55.466,159.886
C03212=1016.957,-67.403,398.437,165.527,55.473,159.887
C03213=1016.951,-67.653,398.448,165.524,55.478,159.887
C03214=1016.946,-67.903,398.458,165.521,55.485,159.888
C03215=1016.941,-68.152,398.468,165.518,55.491,159.888
C03216=1016.935,-68.402,398.478,165.515,55.498,159.889
C03217=1016.930,-68.652,398.487,165.512,55.503,159.889
C03218=1016.925,-68.902,398.498,165.510,55.509,159.890
C03219=1016.920,-69.151,398.507,165.506,55.516,159.890
C03220=1016.915,-69.430,398.519,165.503,55.522,159.890
C03221=1016.909,-69.709,398.530,165.500,55.529,159.891
C03222=1016.903,-69.987,398.541,165.496,55.536,159.891
C03223=1016.897,-70.265,398.553,165.493,55.543,159.892
C03224=1016.892,-70.515,398.563,165.491,55.549,159.892
C03225=1016.887,-70.764,398.573,165.488,55.554,159.893
C03226=1016.882,-71.015,398.583,165.485,55.561,159.893
C03227=1016.877,-71.264,398.593,165.482,55.567,159.894
C03228=1016.871,-71.514,398.603,165.478,55.573,159.894
C03229=1016.867,-71.763,398.613,165.476,55.579,159.894
C03230=1016.861,-72.014,398.623,165.473,55.585,159.895
C03231=1016.856,-72.263,398.633,165.469,55.591,159.895
C03232=1016.851,-72.513,398.643,165.467,55.597,159.896
C03233=1016.846,-72.762,398.653,165.465,55.603,159.896
C03234=1016.841,-73.013,398.663,165.461,55.609,159.896
C03235=1016.836,-73.262,398.673,165.459,55.615,159.897
C03236=1016.831,-73.511,398.683,165.456,55.621,159.897
C03237=1016.826,-73.762,398.693,165.452,55.627,159.897
C03238=1016.821,-74.011,398.703,165.449,55.633,159.898
C03239=1016.815,-74.261,398.713,165.447,55.639,159.898
C03240=1016.811,-74.511,398.722,165.443,55.645,159.899
C03241=1016.805,-74.761,398.732,165.441,55.651,159.899
C03242=1016.801,-75.011,398.742,165.437,55.658,159.900
C03243=1016.795,-75.260,398.751,165.435,55.663,159.900
C03244=1016.790,-75.510,398.761,165.432,55.670,159.900
C03245=1016.785,-75.760,398.770,165.429,55.676,159.901
C03246=1016.779,-76.010,398.780,165.427,55.682,159.901
C03247=1016.774,-76.259,398.790,165.423,55.688,159.902
C03248=1016.769,-76.509,398.799,165.421,55.695,159.902
C03249=1016.764,-76.759,398.809,165.417,55.701,159.903
C03250=1016.758,-77.008,398.818,165.415,55.707,159.903
C03251=1016.753,-77.258,398.828,165.411,55.713,159.903
C03252=1016.748,-77.508,398.837,165.409,55.720,159.904
C03253=1016.743,-77.757,398.847,165.405,55.726,159.904
C03254=1016.737,-78.008,398.857,165.402,55.732,159.905
C03255=1016.733,-78.258,398.866,165.400,55.738,159.905
C03256=1016.728,-78.507,398.876,165.396,55.744,159.905
C03257=1016.722,-78.757,398.885,165.394,55.751,159.906
C03258=1016.717,-79.007,398.894,165.391,55.757,159.906
C03259=1016.713,-79.256,398.904,165.388,55.762,159.907
C03260=1016.706,-79.506,398.914,165.385,55.769,159.907
C03261=1016.702,-79.756,398.923,165.382,55.775,159.908
C03262=1016.697,-80.005,398.933,165.379,55.780,159.908
C03263=1016.691,-80.255,398.942,165.376,55.787,159.908
C03264=1016.686,-80.505,398.951,165.373,55.793,159.909
C03265=1016.681,-80.754,398.960,165.370,55.800,159.909
C03266=1016.676,-81.005,398.970,165.367,55.806,159.910
C03267=1016.670,-81.254,398.979,165.364,55.812,159.910
C03268=1016.666,-81.504,398.988,165.361,55.818,159.910
C03269=1016.660,-81.754,398.997,165.358,55.825,159.911
C03270=1016.655,-82.004,399.007,165.356,55.831,159.912
C03271=1016.650,-82.254,399.015,165.352,55.837,159.912
C03272=1016.645,-82.503,399.025,165.349,55.844,159.912
C03273=1016.640,-82.753,399.034,165.346,55.850,159.913
C03274=1016.633,-83.003,399.043,165.343,55.857,159.913
C03275=1016.629,-83.253,399.052,165.341,55.862,159.913
C03276=1016.624,-83.502,399.061,165.337,55.869,159.914
C03277=1016.619,-83.752,399.070,165.335,55.875,159.914
C03278=1016.613,-84.002,399.079,165.331,55.882,159.915
C03279=1016.608,-84.252,399.088,165.329,55.888,159.915
C03280=1016.603,-84.501,399.098,165.325,55.894,159.915
C03281=1016.597,-84.751,399.106,165.323,55.900,159.916
C03282=1016.593,-85.001,399.116,165.319,55.906,159.916
C03283=1016.587,-85.251,399.125,165.317,55.913,159.917
C03284=1016.581,-85.531,399.134,165.314,55.919,159.917
C03285=1016.576,-85.812,399.145,165.311,55.926,159.918
C03286=1016.570,-86.092,399.155,165.307,55.933,159.918
C03287=1016.564,-86.373,399.165,165.303,55.940,159.919
C03288=1016.559,-86.622,399.175,165.301,55.947,159.919
C03289=1016.554,-86.872,399.183,165.298,55.953,159.920
C03290=1016.549,-87.122,399.192,165.294,55.959,159.920
C03291=1016.543,-87.371,399.201,165.292,55.965,159.920
C03292=1016.538,-87.621,399.210,165.289,55.971,159.921
C03293=1016.533,-87.871,399.219,165.286,55.978,159.921
C03294=1016.528,-88.121,399.228,165.283,55.984,159.921
C03295=1016.523,-88.371,399.238,165.280,55.989,159.922
C03296=1016.518,-88.620,399.246,165.277,55.996,159.922
C03297=1016.512,-88.870,399.255,165.274,56.002,159.923
C03298=1016.508,-89.120,399.264,165.272,56.008,159.923
C03299=1016.502,-89.369,399.273,165.268,56.015,159.923
C03300=1016.498,-89.619,399.282,165.266,56.020,159.924
C03301=1016.493,-89.869,399.290,165.262,56.026,159.924
C03302=1016.487,-90.119,399.299,165.260,56.033,159.925
C03303=1016.482,-90.369,399.308,165.256,56.039,159.925
///RCONF 1,0,0,0,1,0,0,0,0,0,0,0,0,0,0,0,0,0,0,0,0,0,0,0
C03304=1016.477,-90.618,399.318,165.253,56.045,159.925
C03305=1016.472,-90.868,399.327,165.251,56.051,159.926
C03306=1016.467,-91.118,399.335,165.248,56.057,159.926
C03307=1016.462,-91.368,399.344,165.245,56.063,159.927
C03308=1016.457,-91.618,399.353,165.241,56.069,159.927
C03309=1016.452,-91.868,399.361,165.239,56.076,159.927
C03310=1016.447,-92.118,399.370,165.236,56.081,159.928
C03311=1016.442,-92.367,399.380,165.233,56.087,159.928
C03312=1016.437,-92.617,399.389,165.230,56.093,159.928
C03313=1016.432,-92.866,399.397,165.227,56.100,159.929
C03314=1016.427,-93.116,399.406,165.224,56.106,159.929
C03315=1016.422,-93.366,399.415,165.221,56.111,159.930
C03316=1016.417,-93.616,399.423,165.218,56.118,159.930
C03317=1016.412,-93.866,399.432,165.216,56.124,159.930
C03318=1016.407,-94.116,399.441,165.213,56.130,159.931
C03319=1016.402,-94.365,399.449,165.209,56.136,159.931
C03320=1016.397,-94.615,399.458,165.207,56.142,159.931
C03321=1016.392,-94.864,399.467,165.204,56.147,159.932
C03322=1016.386,-95.114,399.476,165.200,56.154,159.932
C03323=1016.382,-95.364,399.485,165.198,56.160,159.933
C03324=1016.377,-95.614,399.494,165.195,56.166,159.933
C03325=1016.372,-95.864,399.503,165.192,56.172,159.933
C03326=1016.367,-96.114,399.511,165.189,56.178,159.933
C03327=1016.362,-96.363,399.520,165.186,56.183,159.934
C03328=1016.357,-96.613,399.529,165.183,56.189,159.934
C03329=1016.352,-96.863,399.537,165.180,56.195,159.934
C03330=1016.347,-97.113,399.546,165.178,56.202,159.935
C03331=1016.342,-97.363,399.555,165.174,56.208,159.935
C03332=1016.337,-97.613,399.563,165.171,56.214,159.936
C03333=1016.332,-97.863,399.572,165.169,56.219,159.936
C03334=1016.327,-98.113,399.580,165.165,56.225,159.936
C03335=1016.323,-98.362,399.588,165.162,56.231,159.937
C03336=1016.317,-98.612,399.597,165.159,56.238,159.937
C03337=1016.312,-98.861,399.605,165.157,56.244,159.937
C03338=1016.307,-99.111,399.614,165.153,56.250,159.938
C03339=1016.303,-99.362,399.622,165.151,56.256,159.938
C03340=1016.297,-99.611,399.630,165.148,56.262,159.939
C03341=1016.292,-99.861,399.639,165.144,56.268,159.939
C03342=1016.287,-100.111,399.647,165.142,56.275,159.939
C03343=1016.282,-100.361,399.655,165.139,56.281,159.940
C03344=1016.277,-100.610,399.663,165.136,56.287,159.940
C03345=1016.272,-100.860,399.672,165.133,56.292,159.940
C03346=1016.267,-101.110,399.680,165.130,56.299,159.941
C03347=1016.262,-101.360,399.688,165.128,56.305,159.941
C03348=1016.256,-101.642,399.698,165.124,56.312,159.942
C03349=1016.251,-101.925,399.708,165.121,56.319,159.942
C03350=1016.245,-102.207,399.716,165.118,56.326,159.943
C03351=1016.240,-102.490,399.726,165.113,56.332,159.943
C03352=1016.234,-102.739,399.734,165.111,56.339,159.943
C03353=1016.229,-102.989,399.743,165.109,56.344,159.944
C03354=1016.224,-103.239,399.751,165.105,56.351,159.944
C03355=1016.220,-103.488,399.759,165.102,56.356,159.944
C03356=1016.214,-103.738,399.767,165.100,56.362,159.945
C03357=1016.209,-103.988,399.775,165.096,56.369,159.945
C03358=1016.204,-104.238,399.783,165.094,56.375,159.945
C03359=1016.199,-104.488,399.792,165.091,56.381,159.946
C03360=1016.195,-104.737,399.799,165.087,56.387,159.946
C03361=1016.189,-104.987,399.808,165.085,56.392,159.946
C03362=1016.185,-105.238,399.816,165.081,56.399,159.946
C03363=1016.180,-105.488,399.825,165.078,56.404,159.947
C03364=1016.175,-105.737,399.833,165.076,56.411,159.947
C03365=1016.170,-105.987,399.841,165.073,56.417,159.948
C03366=1016.165,-106.237,399.849,165.070,56.423,159.948
C03367=1016.160,-106.487,399.857,165.067,56.429,159.948
C03368=1016.155,-106.736,399.865,165.064,56.435,159.949
C03369=1016.150,-106.986,399.873,165.061,56.440,159.949
C03370=1016.145,-107.236,399.881,165.058,56.446,159.949
C03371=1016.141,-107.486,399.889,165.055,56.453,159.950
C03372=1016.135,-107.735,399.897,165.053,56.459,159.950
C03373=1016.130,-107.986,399.905,165.050,56.465,159.951
C03374=1016.126,-108.235,399.913,165.046,56.471,159.951
C03375=1016.121,-108.485,399.921,165.044,56.477,159.951
C03376=1016.116,-108.735,399.929,165.041,56.482,159.951
C03377=1016.110,-108.985,399.936,165.038,56.489,159.952
C03378=1016.106,-109.234,399.944,165.035,56.495,159.952
C03379=1016.100,-109.484,399.952,165.033,56.501,159.953
C03380=1016.095,-109.735,399.960,165.029,56.507,159.953
C03381=1016.091,-109.984,399.967,165.026,56.513,159.953
C03382=1016.086,-110.234,399.976,165.023,56.519,159.953
C03383=1016.081,-110.483,399.983,165.021,56.525,159.954
C03384=1016.076,-110.733,399.992,165.018,56.531,159.954
C03385=1016.071,-110.984,400.000,165.014,56.537,159.955
C03386=1016.066,-111.233,400.006,165.012,56.543,159.955
C03387=1016.061,-111.483,400.015,165.009,56.549,159.955
C03388=1016.056,-111.733,400.023,165.005,56.555,159.955
C03389=1016.051,-111.983,400.030,165.003,56.561,159.956
C03390=1016.046,-112.232,400.039,165.000,56.567,159.956
C03391=1016.042,-112.482,400.046,164.996,56.573,159.956
C03392=1016.037,-112.732,400.054,164.994,56.579,159.957
C03393=1016.032,-112.983,400.062,164.992,56.585,159.957
C03394=1016.026,-113.231,400.069,164.989,56.591,159.958
C03395=1016.021,-113.482,400.077,164.985,56.597,159.958
C03396=1016.017,-113.731,400.084,164.983,56.603,159.958
C03397=1016.012,-113.982,400.092,164.980,56.609,159.959
C03398=1016.008,-114.231,400.100,164.976,56.615,159.959
C03399=1016.003,-114.481,400.108,164.974,56.621,159.959
C03400=1015.998,-114.731,400.115,164.971,56.626,159.960
C03401=1015.993,-114.981,400.122,164.968,56.632,159.960
C03402=1015.987,-115.230,400.131,164.965,56.638,159.960
C03403=1015.983,-115.480,400.138,164.962,56.644,159.960
C03404=1015.978,-115.730,400.146,164.960,56.650,159.961
C03405=1015.973,-115.980,400.153,164.957,56.657,159.961
C03406=1015.968,-116.230,400.161,164.954,56.663,159.962
C03407=1015.964,-116.480,400.168,164.951,56.668,159.962
C03408=1015.959,-116.730,400.176,164.948,56.675,159.962
C03409=1015.953,-116.979,400.183,164.945,56.680,159.963
C03410=1015.948,-117.229,400.191,164.943,56.686,159.963
C03411=1015.944,-117.479,400.199,164.939,56.692,159.963
C03412=1015.938,-117.762,400.207,164.936,56.699,159.964
C03413=1015.933,-118.043,400.215,164.933,56.705,159.964
C03414=1015.927,-118.327,400.224,164.930,56.712,159.964
C03415=1015.922,-118.609,400.232,164.927,56.719,159.965
C03416=1015.917,-118.859,400.239,164.923,56.725,159.965
C03417=1015.912,-119.109,400.247,164.921,56.731,159.965
C03418=1015.908,-119.359,400.254,164.918,56.737,159.966
C03419=1015.902,-119.609,400.261,164.914,56.743,159.966
C03420=1015.898,-119.858,400.269,164.912,56.749,159.966
C03421=1015.893,-120.109,400.276,164.909,56.754,159.967
C03422=1015.888,-120.358,400.283,164.906,56.760,159.967
C03423=1015.883,-120.608,400.291,164.903,56.766,159.967
C03424=1015.878,-120.858,400.298,164.900,56.772,159.968
C03425=1015.873,-121.107,400.305,164.898,56.778,159.968
C03426=1015.868,-121.358,400.313,164.895,56.784,159.968
C03427=1015.864,-121.607,400.320,164.891,56.790,159.968
C03428=1015.858,-121.857,400.327,164.889,56.796,159.969
C03429=1015.854,-122.107,400.335,164.886,56.802,159.969
C03430=1015.850,-122.356,400.342,164.884,56.807,159.970
C03431=1015.844,-122.606,400.349,164.880,56.814,159.970
C03432=1015.840,-122.856,400.357,164.877,56.819,159.970
C03433=1015.835,-123.106,400.364,164.875,56.825,159.970
C03434=1015.830,-123.356,400.371,164.872,56.831,159.971
C03435=1015.825,-123.606,400.378,164.870,56.837,159.971
C03436=1015.821,-123.856,400.386,164.866,56.843,159.971
C03437=1015.815,-124.106,400.393,164.863,56.848,159.971
C03438=1015.811,-124.355,400.400,164.860,56.854,159.972
C03439=1015.806,-124.605,400.407,164.858,56.860,159.972
C03440=1015.801,-124.855,400.415,164.854,56.866,159.972
C03441=1015.797,-125.105,400.421,164.851,56.872,159.973
C03442=1015.792,-125.355,400.428,164.849,56.877,159.973
C03443=1015.787,-125.605,400.436,164.846,56.883,159.973
C03444=1015.782,-125.854,400.443,164.842,56.890,159.974
C03445=1015.778,-126.104,400.449,164.840,56.895,159.974
C03446=1015.772,-126.354,400.457,164.837,56.901,159.974
C03447=1015.768,-126.604,400.464,164.835,56.907,159.975
C03448=1015.763,-126.854,400.470,164.832,56.913,159.975
C03449=1015.759,-127.104,400.478,164.828,56.919,159.975
C03450=1015.753,-127.354,400.485,164.826,56.925,159.976
C03451=1015.749,-127.603,400.492,164.823,56.931,159.976
C03452=1015.744,-127.853,400.498,164.821,56.936,159.976
C03453=1015.739,-128.103,400.505,164.818,56.942,159.977
C03454=1015.734,-128.352,400.512,164.815,56.947,159.977
C03455=1015.730,-128.602,400.521,164.812,56.952,159.977
C03456=1015.727,-128.852,400.529,164.810,56.957,159.977
C03457=1015.723,-129.101,400.538,164.807,56.961,159.977
C03458=1015.720,-129.351,400.548,164.804,56.964,159.977
C03459=1015.718,-129.600,400.558,164.802,56.967,159.977
C03460=1015.715,-129.849,400.569,164.799,56.969,159.976
C03461=1015.714,-130.099,400.581,164.796,56.971,159.976
C03462=1015.712,-130.349,400.593,164.794,56.972,159.976
C03463=1015.711,-130.599,400.605,164.792,56.972,159.975
C03464=1015.710,-130.848,400.618,164.790,56.971,159.975
C03465=1015.709,-131.098,400.633,164.787,56.971,159.974
C03466=1015.710,-131.348,400.647,164.786,56.969,159.973
C03467=1015.710,-131.598,400.662,164.783,56.967,159.972
C03468=1015.710,-131.847,400.678,164.781,56.965,159.971
C03469=1015.712,-132.098,400.694,164.779,56.962,159.970
C03470=1015.713,-132.347,400.711,164.778,56.959,159.969
C03471=1015.715,-132.596,400.728,164.775,56.954,159.968
C03472=1015.718,-132.846,400.747,164.774,56.950,159.966
C03473=1015.721,-133.095,400.765,164.771,56.945,159.965
C03474=1015.723,-133.345,400.784,164.770,56.939,159.963
C03475=1015.726,-133.594,400.804,164.767,56.932,159.962
C03476=1015.480,-133.621,400.405,164.734,57.301,160.019
C03477=1015.477,-133.371,400.385,164.735,57.308,160.020
C03478=1015.473,-133.123,400.366,164.737,57.314,160.022
C03479=1015.471,-132.872,400.347,164.739,57.319,160.023
C03480=1015.469,-132.622,400.329,164.741,57.323,160.024
C03481=1015.467,-132.372,400.311,164.743,57.327,160.026
C03482=1015.465,-132.124,400.295,164.745,57.331,160.027
C03483=1015.464,-131.873,400.278,164.747,57.334,160.028
C03484=1015.463,-131.624,400.263,164.749,57.337,160.029
C03485=1015.463,-131.374,400.248,164.751,57.338,160.030
C03486=1015.463,-131.125,400.233,164.753,57.340,160.031
C03487=1015.464,-130.875,400.219,164.756,57.340,160.032
C03488=1015.464,-130.625,400.206,164.757,57.341,160.032
C03489=1015.465,-130.375,400.193,164.760,57.340,160.033
C03490=1015.467,-130.125,400.181,164.762,57.339,160.033
C03491=1015.469,-129.876,400.169,164.765,57.338,160.034
C03492=1015.471,-129.626,400.159,164.767,57.335,160.034
C03493=1015.473,-129.377,400.148,164.770,57.333,160.034
C03494=1015.477,-129.127,400.139,164.772,57.329,160.034
C03495=1015.480,-128.877,400.130,164.774,57.326,160.034
C03496=1015.484,-128.628,400.121,164.778,57.321,160.034
C03497=1015.488,-128.379,400.114,164.780,57.317,160.034
C03498=1015.492,-128.129,400.106,164.783,57.312,160.034
C03499=1015.497,-127.879,400.099,164.786,57.305,160.033
C03500=1015.502,-127.630,400.092,164.789,57.299,160.033
C03501=1015.506,-127.380,400.085,164.791,57.294,160.033
C03502=1015.511,-127.130,400.078,164.794,57.288,160.032
C03503=1015.516,-126.880,400.071,164.796,57.282,160.032
C03504=1015.521,-126.630,400.065,164.800,57.276,160.032
C03505=1015.525,-126.380,400.057,164.803,57.270,160.031
C03506=1015.530,-126.131,400.050,164.805,57.264,160.031
C03507=1015.535,-125.880,400.043,164.808,57.258,160.031
C03508=1015.540,-125.631,400.037,164.811,57.252,160.030
C03509=1015.544,-125.381,400.029,164.814,57.246,160.030
C03510=1015.549,-125.132,400.022,164.816,57.240,160.030
C03511=1015.554,-124.881,400.015,164.819,57.234,160.029
C03512=1015.559,-124.632,400.008,164.823,57.228,160.029
C03513=1015.563,-124.382,400.001,164.825,57.222,160.029
C03514=1015.569,-124.132,399.994,164.828,57.216,160.028
C03515=1015.573,-123.882,399.987,164.830,57.211,160.028
C03516=1015.578,-123.632,399.980,164.834,57.205,160.028
C03517=1015.583,-123.382,399.973,164.837,57.199,160.028
C03518=1015.588,-123.132,399.965,164.839,57.193,160.027
C03519=1015.592,-122.883,399.958,164.842,57.188,160.027
C03520=1015.597,-122.633,399.951,164.846,57.181,160.027
C03521=1015.602,-122.383,399.944,164.848,57.176,160.026
C03522=1015.606,-122.133,399.937,164.851,57.170,160.026
C03523=1015.612,-121.883,399.929,164.853,57.164,160.026
C03524=1015.616,-121.633,399.922,164.857,57.158,160.026
C03525=1015.621,-121.384,399.915,164.859,57.152,160.025
C03526=1015.626,-121.134,399.907,164.862,57.146,160.025
C03527=1015.631,-120.884,399.900,164.864,57.140,160.024
C03528=1015.635,-120.634,399.893,164.868,57.134,160.024
C03529=1015.641,-120.384,399.885,164.871,57.128,160.024
C03530=1015.645,-120.135,399.878,164.873,57.122,160.024
C03531=1015.649,-119.885,399.871,164.877,57.116,160.023
C03532=1015.655,-119.635,399.863,164.879,57.110,160.023
C03533=1015.659,-119.385,399.857,164.882,57.104,160.023
C03534=1015.664,-119.134,399.849,164.885,57.099,160.022
C03535=1015.669,-118.885,399.842,164.888,57.092,160.022
C03536=1015.674,-118.635,399.834,164.891,57.087,160.022
C03537=1015.680,-118.353,399.826,164.894,57.080,160.021
C03538=1015.685,-118.071,399.818,164.897,57.073,160.021
C03539=1015.691,-117.788,399.809,164.900,57.066,160.020
C03540=1015.695,-117.505,399.801,164.904,57.059,160.020
C03541=1015.700,-117.256,399.794,164.906,57.054,160.020
C03542=1015.705,-117.006,399.786,164.910,57.047,160.020
C03543=1015.710,-116.756,399.779,164.912,57.041,160.019
C03544=1015.715,-116.506,399.770,164.914,57.035,160.019
C03545=1015.720,-116.257,399.763,164.918,57.029,160.018
C03546=1015.725,-116.007,399.756,164.920,57.023,160.018
C03547=1015.729,-115.757,399.748,164.923,57.017,160.018
C03548=1015.734,-115.507,399.740,164.927,57.011,160.017
C03549=1015.739,-115.257,399.734,164.929,57.005,160.017
C03550=1015.744,-115.007,399.726,164.932,56.999,160.017
C03551=1015.749,-114.757,399.718,164.935,56.993,160.017
C03552=1015.754,-114.507,399.711,164.938,56.987,160.016
C03553=1015.758,-114.258,399.703,164.941,56.981,160.016
C03554=1015.764,-114.008,399.695,164.944,56.974,160.015
C03555=1015.768,-113.758,399.688,164.946,56.969,160.015
C03556=1015.773,-113.508,399.680,164.949,56.963,160.015
C03557=1015.778,-113.259,399.672,164.952,56.957,160.014
C03558=1015.783,-113.009,399.664,164.955,56.951,160.014
C03559=1015.787,-112.759,399.657,164.958,56.945,160.014
C03560=1015.792,-112.509,399.649,164.961,56.939,160.013
C03561=1015.797,-112.260,399.641,164.964,56.933,160.013
C03562=1015.803,-112.010,399.634,164.966,56.927,160.013
C03563=1015.808,-111.759,399.626,164.970,56.921,160.012
C03564=1015.812,-111.510,399.619,164.972,56.914,160.012
C03565=1015.817,-111.260,399.610,164.975,56.909,160.011
C03566=1015.822,-111.010,399.603,164.978,56.902,160.011
C03567=1015.827,-110.760,399.595,164.981,56.897,160.011
C03568=1015.832,-110.510,399.586,164.984,56.890,160.011
C03569=1015.836,-110.261,399.579,164.987,56.884,160.010
C03570=1015.842,-110.011,399.572,164.990,56.879,160.010
C03571=1015.846,-109.761,399.565,164.993,56.872,160.010
C03572=1015.852,-109.511,399.556,164.995,56.866,160.009
C03573=1015.857,-109.261,399.548,164.999,56.860,160.009
C03574=1015.861,-109.012,399.540,165.001,56.854,160.009
C03575=1015.866,-108.762,399.532,165.003,56.847,160.008
C03576=1015.871,-108.511,399.525,165.007,56.841,160.008
C03577=1015.876,-108.262,399.516,165.010,56.835,160.007
C03578=1015.881,-108.012,399.509,165.013,56.829,160.007
C03579=1015.886,-107.762,399.501,165.016,56.823,160.007
C03580=1015.890,-107.513,399.493,165.018,56.817,160.006
C03581=1015.895,-107.262,399.485,165.022,56.811,160.006
C03582=1015.901,-107.013,399.477,165.024,56.805,160.006
C03583=1015.905,-106.763,399.469,165.027,56.799,160.005
C03584=1015.910,-106.513,399.461,165.030,56.793,160.005
C03585=1015.915,-106.263,399.453,165.033,56.787,160.005
C03586=1015.920,-106.014,399.445,165.036,56.780,160.004
C03587=1015.925,-105.764,399.437,165.039,56.774,160.004
C03588=1015.930,-105.514,399.429,165.041,56.769,160.003
C03589=1015.934,-105.264,399.421,165.045,56.762,160.003
C03590=1015.940,-105.014,399.413,165.047,56.757,160.003
C03591=1015.945,-104.765,399.404,165.051,56.750,160.003
C03592=1015.950,-104.514,399.396,165.053,56.744,160.002
C03593=1015.955,-104.265,399.388,165.056,56.738,160.002
C03594=1015.959,-104.015,399.381,165.059,56.732,160.001
C03595=1015.965,-103.765,399.372,165.062,56.726,160.001
C03596=1015.970,-103.515,399.364,165.066,56.720,160.001
C03597=1015.974,-103.266,399.356,165.068,56.713,160.000
C03598=1015.979,-103.016,399.347,165.070,56.708,160.000
C03599=1015.984,-102.766,399.339,165.074,56.701,160.000
C03600=1015.989,-102.516,399.331,165.077,56.696,159.999
C03601=1015.995,-102.234,399.322,165.080,56.689,159.999
C03602=1016.000,-101.952,399.312,165.083,56.682,159.998
C03603=1016.006,-101.669,399.303,165.087,56.674,159.998
C03604=1016.011,-101.387,399.294,165.090,56.667,159.998
C03605=1016.016,-101.138,399.285,165.093,56.662,159.997
C03606=1016.021,-100.887,399.278,165.096,56.655,159.997
C03607=1016.027,-100.638,399.269,165.098,56.649,159.996
C03608=1016.032,-100.388,399.261,165.102,56.643,159.996
C03609=1016.037,-100.139,399.253,165.104,56.636,159.996
C03610=1016.042,-99.888,399.245,165.107,56.630,159.995
C03611=1016.046,-99.638,399.236,165.110,56.624,159.995
C03612=1016.051,-99.389,399.227,165.112,56.618,159.994
C03613=1016.057,-99.139,399.219,165.116,56.612,159.994
C03614=1016.062,-98.889,399.211,165.119,56.606,159.994
C03615=1016.066,-98.640,399.203,165.122,56.599,159.993
C03616=1016.071,-98.390,399.194,165.124,56.593,159.993
C03617=1016.077,-98.140,399.186,165.128,56.587,159.993
C03618=1016.082,-97.890,399.178,165.130,56.580,159.992
C03619=1016.086,-97.640,399.169,165.134,56.574,159.992
C03620=1016.091,-97.390,399.161,165.136,56.569,159.991
C03621=1016.096,-97.140,399.151,165.139,56.563,159.991
C03622=1016.101,-96.890,399.143,165.143,56.557,159.991
C03623=1016.107,-96.641,399.135,165.145,56.551,159.990
C03624=1016.111,-96.391,399.125,165.147,56.544,159.990
C03625=1016.116,-96.141,399.117,165.151,56.538,159.990
C03626=1016.120,-95.892,399.108,165.154,56.532,159.989
C03627=1016.126,-95.642,399.100,165.157,56.526,159.989
C03628=1016.131,-95.392,399.091,165.160,56.520,159.989
C03629=1016.135,-95.142,399.082,165.162,56.514,159.988
